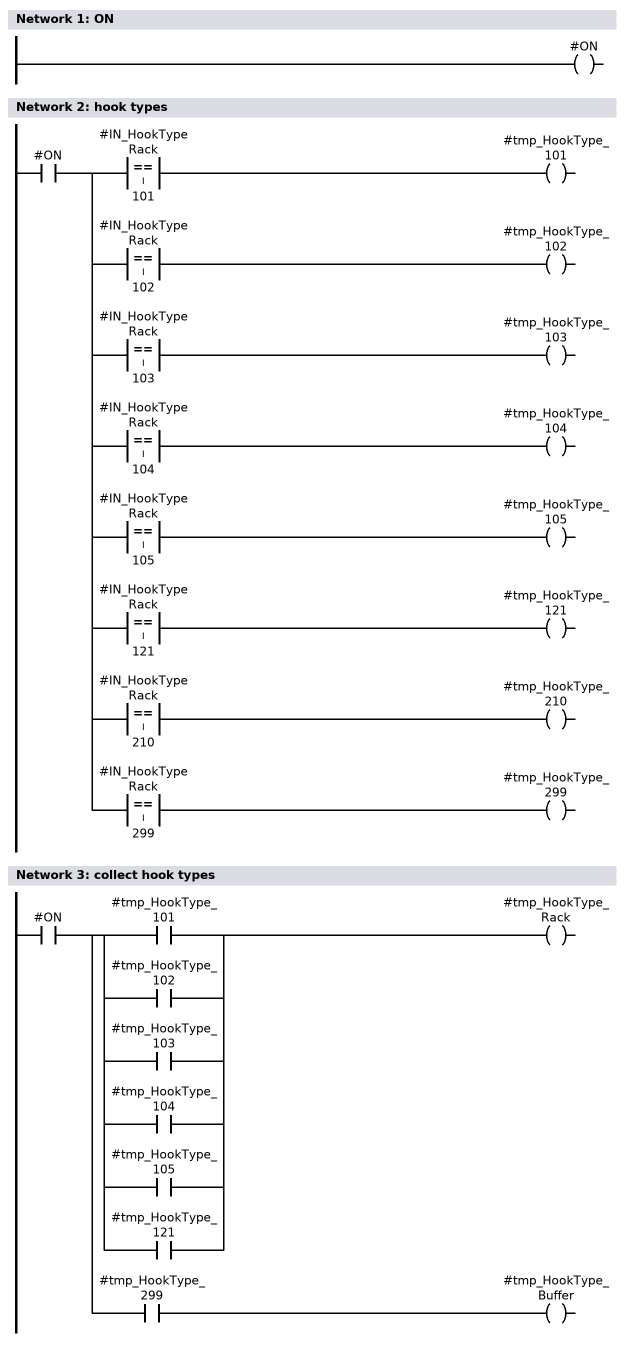
[picture p237: CheckHookType networks 1-3]
NETWORK
TITLE = ON
      SET;
      =     #ON;
NETWORK
TITLE = hook types
      A     #ON;
      =     L 7.0;
      A     L 7.0;
      A(;
      L     #IN_HookTypeRack;
      L     101;
      ==I;
      );
      =     #tmp_HookType_101;
      A     L 7.0;
      A(;
      L     #IN_HookTypeRack;
      L     102;
      ==I;
      );
      =     #tmp_HookType_102;
      A     L 7.0;
      A(;
      L     #IN_HookTypeRack;
      L     103;
      ==I;
      );
      =     #tmp_HookType_103;
      A     L 7.0;
      A(;
      L     #IN_HookTypeRack;
      L     104;
      ==I;
      );
      =     #tmp_HookType_104;
      A     L 7.0;
      A(;
      L     #IN_HookTypeRack;
      L     105;
      ==I;
      );
      =     #tmp_HookType_105;
      A     L 7.0;
      A(;
      L     #IN_HookTypeRack;
      L     121;
      ==I;
      );
      =     #tmp_HookType_121;
      A     L 7.0;
      A(;
      L     #IN_HookTypeRack;
      L     210;
      ==I;
      );
      =     #tmp_HookType_210;
      A     L 7.0;
      A(;
      L     #IN_HookTypeRack;
      L     299;
      ==I;
      );
      =     #tmp_HookType_299;
NETWORK
TITLE = collect hook types
      A     #ON;
      =     L 7.0;
      A     L 7.0;
      A(;
      O     #tmp_HookType_101;
      O     #tmp_HookType_102;
      O     #tmp_HookType_103;
      O     #tmp_HookType_104;
      O     #tmp_HookType_105;
      O     #tmp_HookType_121;
      );
      =     #tmp_HookType_Rack;
      A     L 7.0;
      A     #tmp_HookType_299;
      =     #tmp_HookType_Buffer;
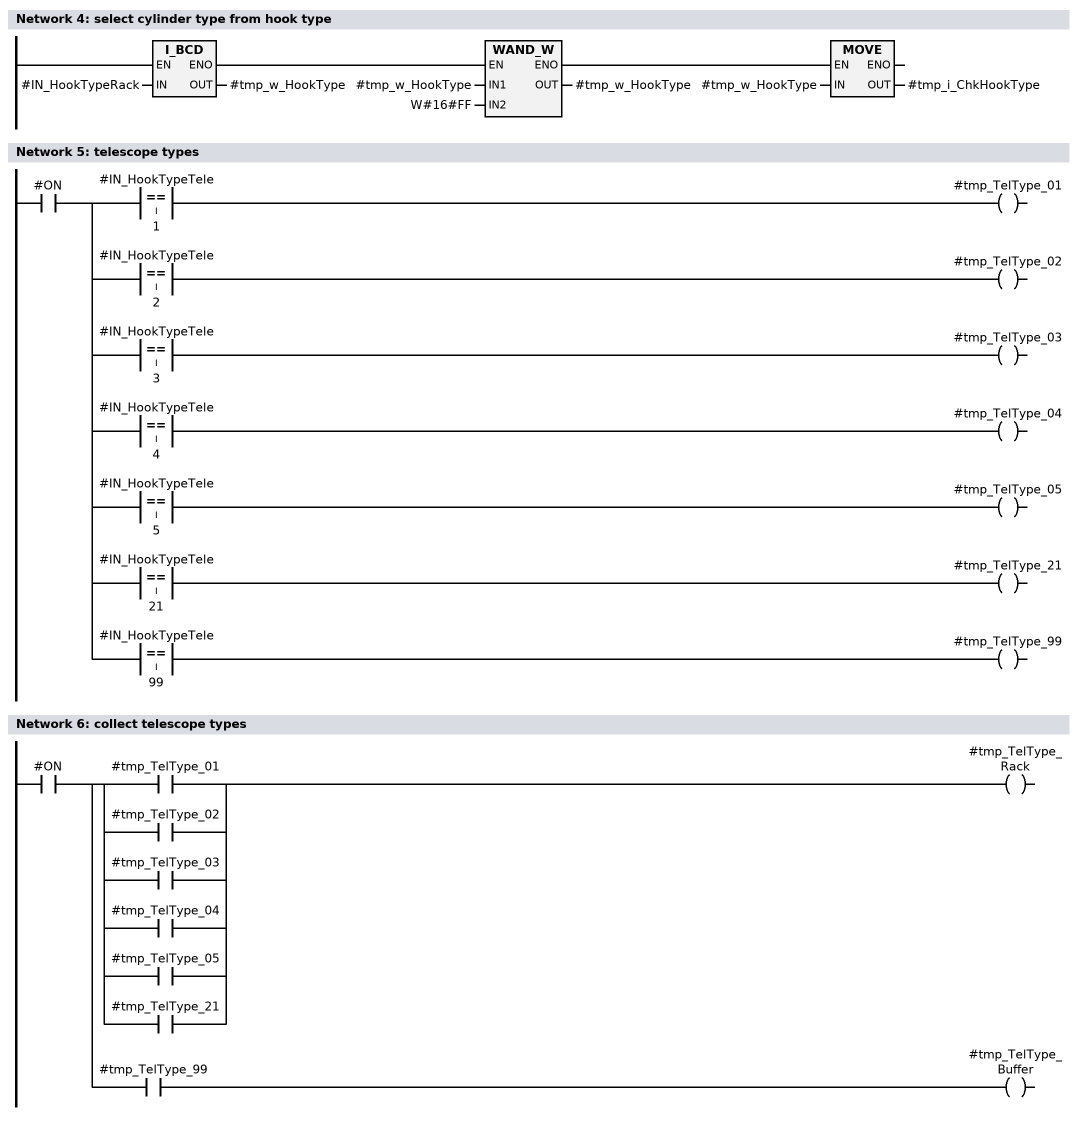
NETWORK
TITLE = select cylinder type from hook type
      A(;
      A(;
      L     #IN_HookTypeRack;
      ITB;
      T     #tmp_w_HookType;
      AN    OV;
      SAVE;
      CLR;
      A     BR;
      );
      JNB   _001;
      L     #tmp_w_HookType;
      L     W#16#FF;
      AW;
      T     #tmp_w_HookType;
      SET;
      SAVE;
      CLR;
_001: A     BR;
      );
      JNB   _002;
      L     #tmp_w_HookType;
      T     #tmp_i_ChkHookType;
_002: NOP   0;
NETWORK
TITLE = telescope types
      A     #ON;
      =     L 7.0;
      A     L 7.0;
      A(;
      L     #IN_HookTypeTele;
      L     1;
      ==I;
      );
      =     #tmp_TelType_01;
      A     L 7.0;
      A(;
      L     #IN_HookTypeTele;
      L     2;
      ==I;
      );
      =     #tmp_TelType_02;
      A     L 7.0;
      A(;
      L     #IN_HookTypeTele;
      L     3;
      ==I;
      );
      =     #tmp_TelType_03;
      A     L 7.0;
      A(;
      L     #IN_HookTypeTele;
      L     4;
      ==I;
      );
      =     #tmp_TelType_04;
      A     L 7.0;
      A(;
      L     #IN_HookTypeTele;
      L     5;
      ==I;
      );
      =     #tmp_TelType_05;
      A     L 7.0;
      A(;
      L     #IN_HookTypeTele;
      L     21;
      ==I;
      );
      =     #tmp_TelType_21;
      A     L 7.0;
      A(;
      L     #IN_HookTypeTele;
      L     99;
      ==I;
      );
      =     #tmp_TelType_99;
NETWORK
TITLE = collect telescope types
      A     #ON;
      =     L 7.0;
      A     L 7.0;
      A(;
      O     #tmp_TelType_01;
      O     #tmp_TelType_02;
      O     #tmp_TelType_03;
      O     #tmp_TelType_04;
      O     #tmp_TelType_05;
      O     #tmp_TelType_21;
      );
      =     #tmp_TelType_Rack;
      A     L 7.0;
      A     #tmp_TelType_99;
      =     #tmp_TelType_Buffer;
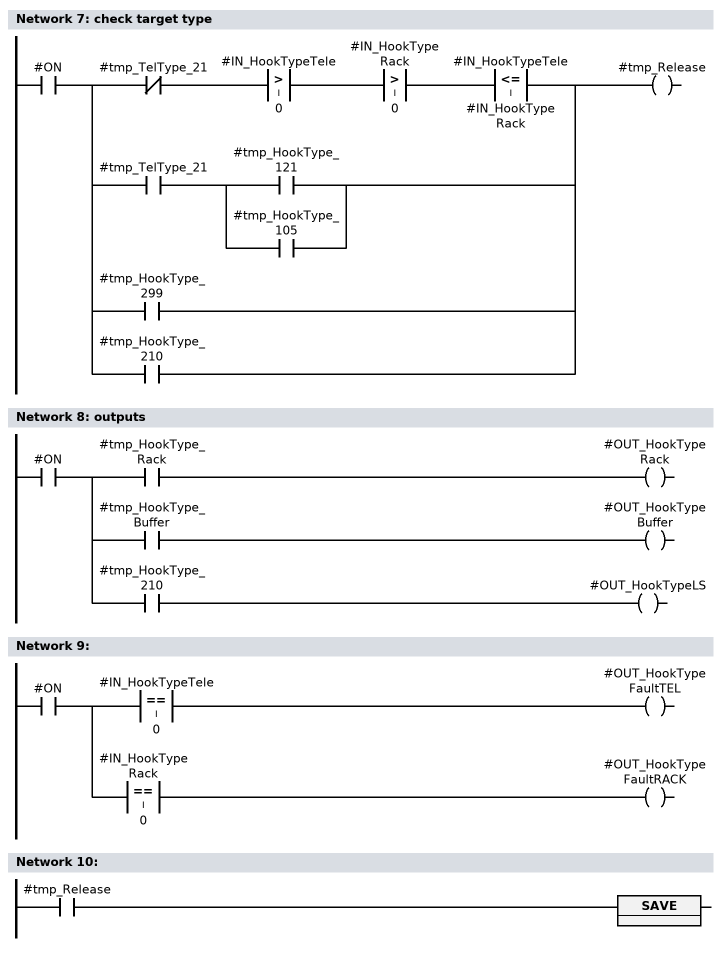
NETWORK
TITLE = check target type
      A     #ON;
      A(;
      AN    #tmp_TelType_21;
      A(;
      L     #IN_HookTypeTele;
      L     0;
      >I;
      );
      A(;
      L     #IN_HookTypeRack;
      L     0;
      >I;
      );
      A(;
      L     #IN_HookTypeTele;
      L     #IN_HookTypeRack;
      <=I;
      );
      O;
      A     #tmp_TelType_21;
      A(;
      O     #tmp_HookType_121;
      O     #tmp_HookType_105;
      );
      O     #tmp_HookType_299;
      O     #tmp_HookType_210;
      );
      =     #tmp_Release;
NETWORK
TITLE = outputs
      A     #ON;
      =     L 7.0;
      A     L 7.0;
      A     #tmp_HookType_Rack;
      =     #OUT_HookTypeRack;
      A     L 7.0;
      A     #tmp_HookType_Buffer;
      =     #OUT_HookTypeBuffer;
      A     L 7.0;
      A     #tmp_HookType_210;
      =     #OUT_HookTypeLS;
NETWORK
TITLE =
      A     #ON;
      =     L 7.0;
      A     L 7.0;
      A(;
      L     #IN_HookTypeTele;
      L     0;
      ==I;
      );
      =     #OUT_HookTypeFaultTEL;
      A     L 7.0;
      A(;
      L     #IN_HookTypeRack;
      L     0;
      ==I;
      );
      =     #OUT_HookTypeFaultRACK;
NETWORK
TITLE =
      A     #tmp_Release;
      SAVE;
END_FUNCTION

FUNCTION "CheckWindowDi" : VOID	// FC 100
TITLE = Check Window
VERSION : 1.0
VAR_INPUT
  IN_diValue : DINT ;
  IN_diTestFor : DINT ;
  IN_diTolMinus : DINT ;
  IN_diTolPlus : DINT ;
END_VAR
VAR_OUTPUT
  OUT_xInWindow : BOOL ;
  OUT_udiAbsDiff : DINT ;
END_VAR
VAR_TEMP
  INT_diWinMinus : DINT ;
  INT_diWinPlus : DINT ;
  INT_xInWindow : BOOL ;
END_VAR
BEGIN
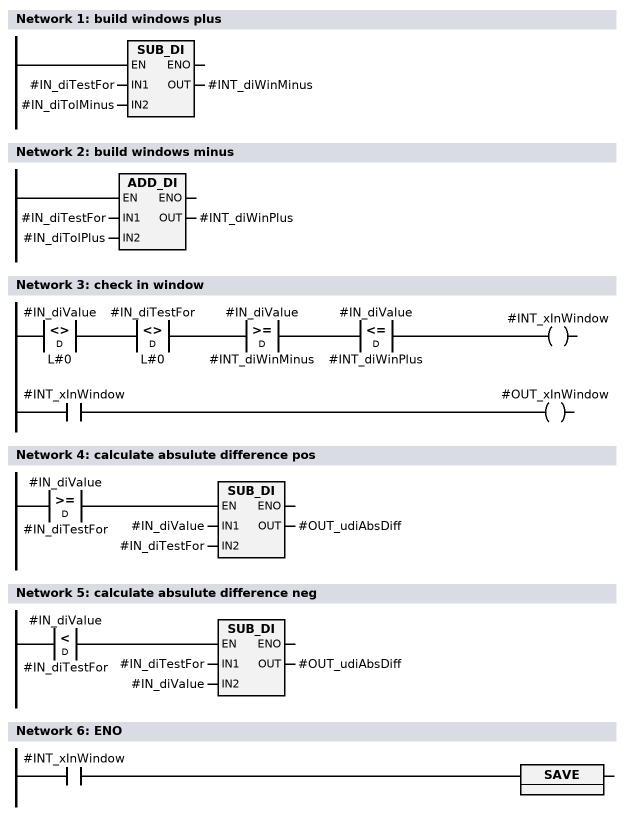
NETWORK
TITLE = build windows plus
      L     #IN_diTestFor;
      L     #IN_diTolMinus;
      -D;
      T     #INT_diWinMinus;
      NOP   0;
NETWORK
TITLE = build windows minus
      L     #IN_diTestFor;
      L     #IN_diTolPlus;
      +D;
      T     #INT_diWinPlus;
      NOP   0;
NETWORK
TITLE = check in window
      A(;
      L     #IN_diValue;
      L     L#0;
      <>D;
      );
      A(;
      L     #IN_diTestFor;
      L     L#0;
      <>D;
      );
      A(;
      L     #IN_diValue;
      L     #INT_diWinMinus;
      >=D;
      );
      A(;
      L     #IN_diValue;
      L     #INT_diWinPlus;
      <=D;
      );
      =     #INT_xInWindow;
      A     #INT_xInWindow;
      =     #OUT_xInWindow;
NETWORK
TITLE = calculate absulute difference pos
      A(;
      L     #IN_diValue;
      L     #IN_diTestFor;
      >=D;
      );
      JNB   _001;
      L     #IN_diValue;
      L     #IN_diTestFor;
      -D;
      T     #OUT_udiAbsDiff;
_001: NOP   0;
NETWORK
TITLE = calculate absulute difference neg
      A(;
      L     #IN_diValue;
      L     #IN_diTestFor;
      <D;
      );
      JNB   _002;
      L     #IN_diTestFor;
      L     #IN_diValue;
      -D;
      T     #OUT_udiAbsDiff;
_002: NOP   0;
NETWORK
TITLE = ENO
      A     #INT_xInWindow;
      SAVE;
END_FUNCTION

FUNCTION "Communication" : VOID	// FC 103
VERSION : 0.1
VAR_TEMP
  tmp_result : INT ;
  rel_online : BOOL ;
  val : DINT ;
END_VAR
BEGIN
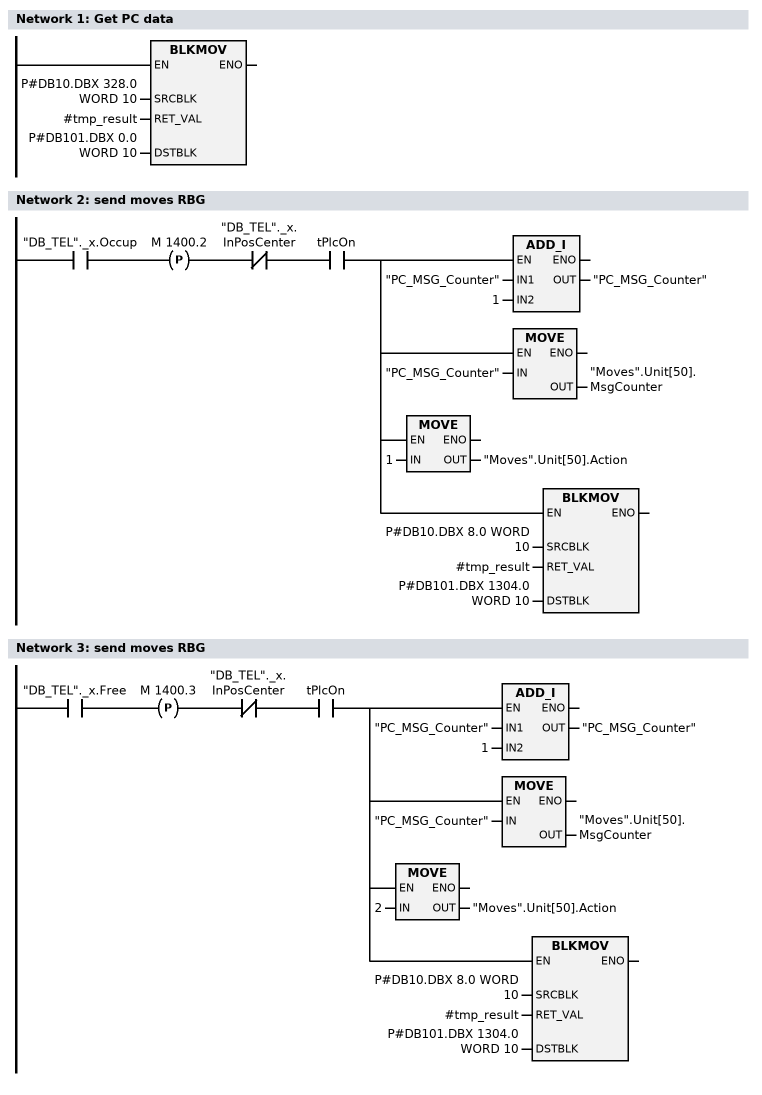
NETWORK
TITLE = Get PC data
      CALL  "BLKMOV" (
           SRCBLK                   := P#DB10.DBX 328.0 WORD 10,
           RET_VAL                  := #tmp_result,
           DSTBLK                   := P#DB101.DBX 0.0 WORD 10);
      NOP   0;
NETWORK
TITLE = send moves RBG
//Telescopes occupied
      A     "DB_TEL"._x.Occup;
      FP    M 1400.2;
      AN    "DB_TEL"._x.InPosCenter;
      A     "tPlcOn";
      =     L 8.0;
      A     L 8.0;
      JNB   _001;
      L     "PC_MSG_Counter";
      L     1;
      +I;
      T     "PC_MSG_Counter";
_001: NOP   0;
      A     L 8.0;
      JNB   _002;
      L     "PC_MSG_Counter";
      T     "Moves".Unit[50].MsgCounter;
_002: NOP   0;
      A     L 8.0;
      JNB   _003;
      L     1;
      T     "Moves".Unit[50].Action;
_003: NOP   0;
      A     L 8.0;
      JNB   _004;
      CALL  "BLKMOV" (
           SRCBLK                   := P#DB10.DBX 8.0 WORD 10,
           RET_VAL                  := #tmp_result,
           DSTBLK                   := P#DB101.DBX 1304.0 WORD 10);
_004: NOP   0;
NETWORK
TITLE = send moves RBG
//Telescopes empty
      A     "DB_TEL"._x.Free;
      FP    M 1400.3;
      AN    "DB_TEL"._x.InPosCenter;
      A     "tPlcOn";
      =     L 8.0;
      A     L 8.0;
      JNB   _005;
      L     "PC_MSG_Counter";
      L     1;
      +I;
      T     "PC_MSG_Counter";
_005: NOP   0;
      A     L 8.0;
      JNB   _006;
      L     "PC_MSG_Counter";
      T     "Moves".Unit[50].MsgCounter;
_006: NOP   0;
      A     L 8.0;
      JNB   _007;
      L     2;
      T     "Moves".Unit[50].Action;
_007: NOP   0;
      A     L 8.0;
      JNB   _008;
      CALL  "BLKMOV" (
           SRCBLK                   := P#DB10.DBX 8.0 WORD 10,
           RET_VAL                  := #tmp_result,
           DSTBLK                   := P#DB101.DBX 1304.0 WORD 10);
_008: NOP   0;
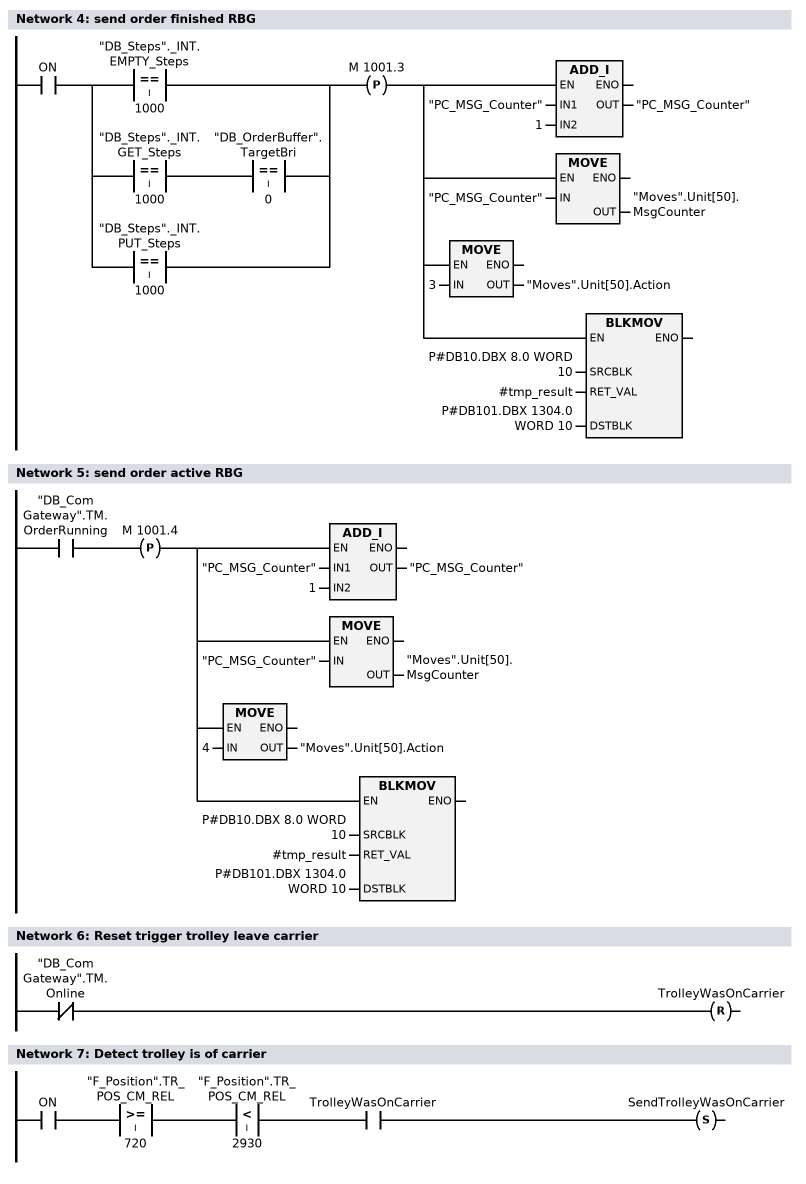
NETWORK
TITLE = send order finished RBG
      A     "ON";
      A(;
      O(;
      L     "DB_Steps"._INT.EMPTY_Steps;
      L     1000;
      ==I;
      );
      O;
      A(;
      L     "DB_Steps"._INT.GET_Steps;
      L     1000;
      ==I;
      );
      A(;
      L     "DB_OrderBuffer".TargetBri;
      L     0;
      ==I;
      );
      O(;
      L     "DB_Steps"._INT.PUT_Steps;
      L     1000;
      ==I;
      );
      );
      FP    M 1001.3;
      =     L 8.0;
      A     L 8.0;
      JNB   _009;
      L     "PC_MSG_Counter";
      L     1;
      +I;
      T     "PC_MSG_Counter";
_009: NOP   0;
      A     L 8.0;
      JNB   _00a;
      L     "PC_MSG_Counter";
      T     "Moves".Unit[50].MsgCounter;
_00a: NOP   0;
      A     L 8.0;
      JNB   _00b;
      L     3;
      T     "Moves".Unit[50].Action;
_00b: NOP   0;
      A     L 8.0;
      JNB   _00c;
      CALL  "BLKMOV" (
           SRCBLK                   := P#DB10.DBX 8.0 WORD 10,
           RET_VAL                  := #tmp_result,
           DSTBLK                   := P#DB101.DBX 1304.0 WORD 10);
_00c: NOP   0;
NETWORK
TITLE = send order active RBG
      A     "DB_ComGateway".TM.OrderRunning;
      FP    M 1001.4;
      =     L 8.0;
      A     L 8.0;
      JNB   _00d;
      L     "PC_MSG_Counter";
      L     1;
      +I;
      T     "PC_MSG_Counter";
_00d: NOP   0;
      A     L 8.0;
      JNB   _00e;
      L     "PC_MSG_Counter";
      T     "Moves".Unit[50].MsgCounter;
_00e: NOP   0;
      A     L 8.0;
      JNB   _00f;
      L     4;
      T     "Moves".Unit[50].Action;
_00f: NOP   0;
      A     L 8.0;
      JNB   _010;
      CALL  "BLKMOV" (
           SRCBLK                   := P#DB10.DBX 8.0 WORD 10,
           RET_VAL                  := #tmp_result,
           DSTBLK                   := P#DB101.DBX 1304.0 WORD 10);
_010: NOP   0;
NETWORK
TITLE = Reset trigger trolley leave carrier
      AN    "DB_ComGateway".TM.Online;
      R     "TrolleyWasOnCarrier";
NETWORK
TITLE = Detect trolley is of carrier
      A     "ON";
      A(;
      L     "F_Position".TR_POS_CM_REL;
      L     720;
      >=I;
      );
      A(;
      L     "F_Position".TR_POS_CM_REL;
      L     2930;
      <I;
      );
      A     "TrolleyWasOnCarrier";
      S     "SendTrolleyWasOnCarrier";
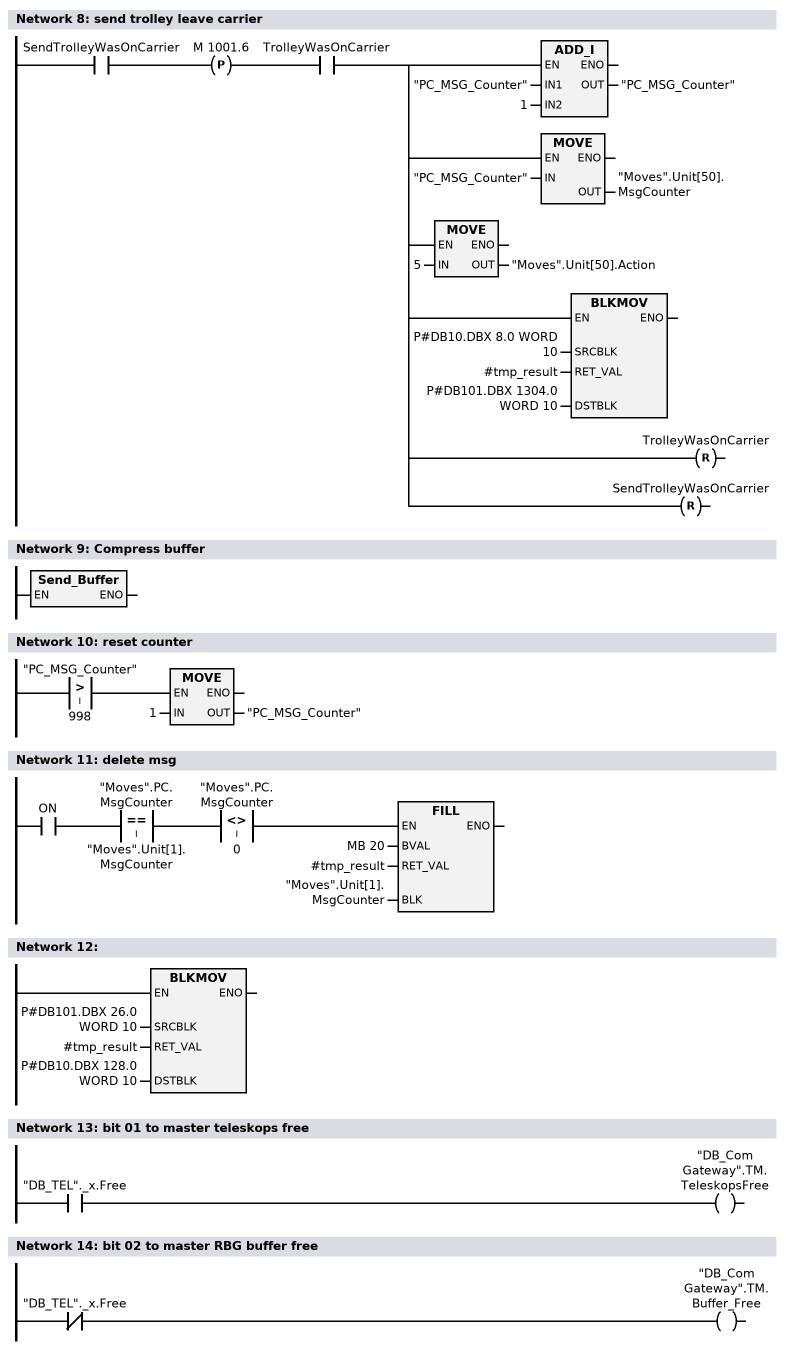
NETWORK
TITLE = send trolley leave carrier
      A     "SendTrolleyWasOnCarrier";
      FP    M 1001.6;
      A     "TrolleyWasOnCarrier";
      =     L 8.0;
      A     L 8.0;
      JNB   _011;
      L     "PC_MSG_Counter";
      L     1;
      +I;
      T     "PC_MSG_Counter";
_011: NOP   0;
      A     L 8.0;
      JNB   _012;
      L     "PC_MSG_Counter";
      T     "Moves".Unit[50].MsgCounter;
_012: NOP   0;
      A     L 8.0;
      JNB   _013;
      L     5;
      T     "Moves".Unit[50].Action;
_013: NOP   0;
      A     L 8.0;
      JNB   _014;
      CALL  "BLKMOV" (
           SRCBLK                   := P#DB10.DBX 8.0 WORD 10,
           RET_VAL                  := #tmp_result,
           DSTBLK                   := P#DB101.DBX 1304.0 WORD 10);
_014: NOP   0;
      A     L 8.0;
      BLD   102;
      R     "TrolleyWasOnCarrier";
      A     L 8.0;
      BLD   102;
      R     "SendTrolleyWasOnCarrier";
NETWORK
TITLE = Compress buffer
      CALL  "Send_Buffer";
      NOP   0;
NETWORK
TITLE = reset counter
      A(;
      L     "PC_MSG_Counter";
      L     998;
      >I;
      );
      JNB   _015;
      L     1;
      T     "PC_MSG_Counter";
_015: NOP   0;
NETWORK
TITLE = delete msg
      A     "ON";
      A(;
      L     "Moves".PC.MsgCounter;
      L     "Moves".Unit[1].MsgCounter;
      ==I;
      );
      A(;
      L     "Moves".PC.MsgCounter;
      L     0;
      <>I;
      );
      JNB   _016;
      CALL  "FILL" (
           BVAL                     := MB 20,
           RET_VAL                  := #tmp_result,
           BLK                      := "Moves".Unit[1].MsgCounter);
_016: NOP   0;
NETWORK
TITLE =
      CALL  "BLKMOV" (
           SRCBLK                   := P#DB101.DBX 26.0 WORD 10,
           RET_VAL                  := #tmp_result,
           DSTBLK                   := P#DB10.DBX 128.0 WORD 10);
      NOP   0;
NETWORK
TITLE = bit 01 to master teleskops free
      A     "DB_TEL"._x.Free;
      =     "DB_ComGateway".TM.TeleskopsFree;
NETWORK
TITLE = bit 02 to master RBG buffer free
      AN    "DB_TEL"._x.Free;
      =     "DB_ComGateway".TM.Buffer_Free;
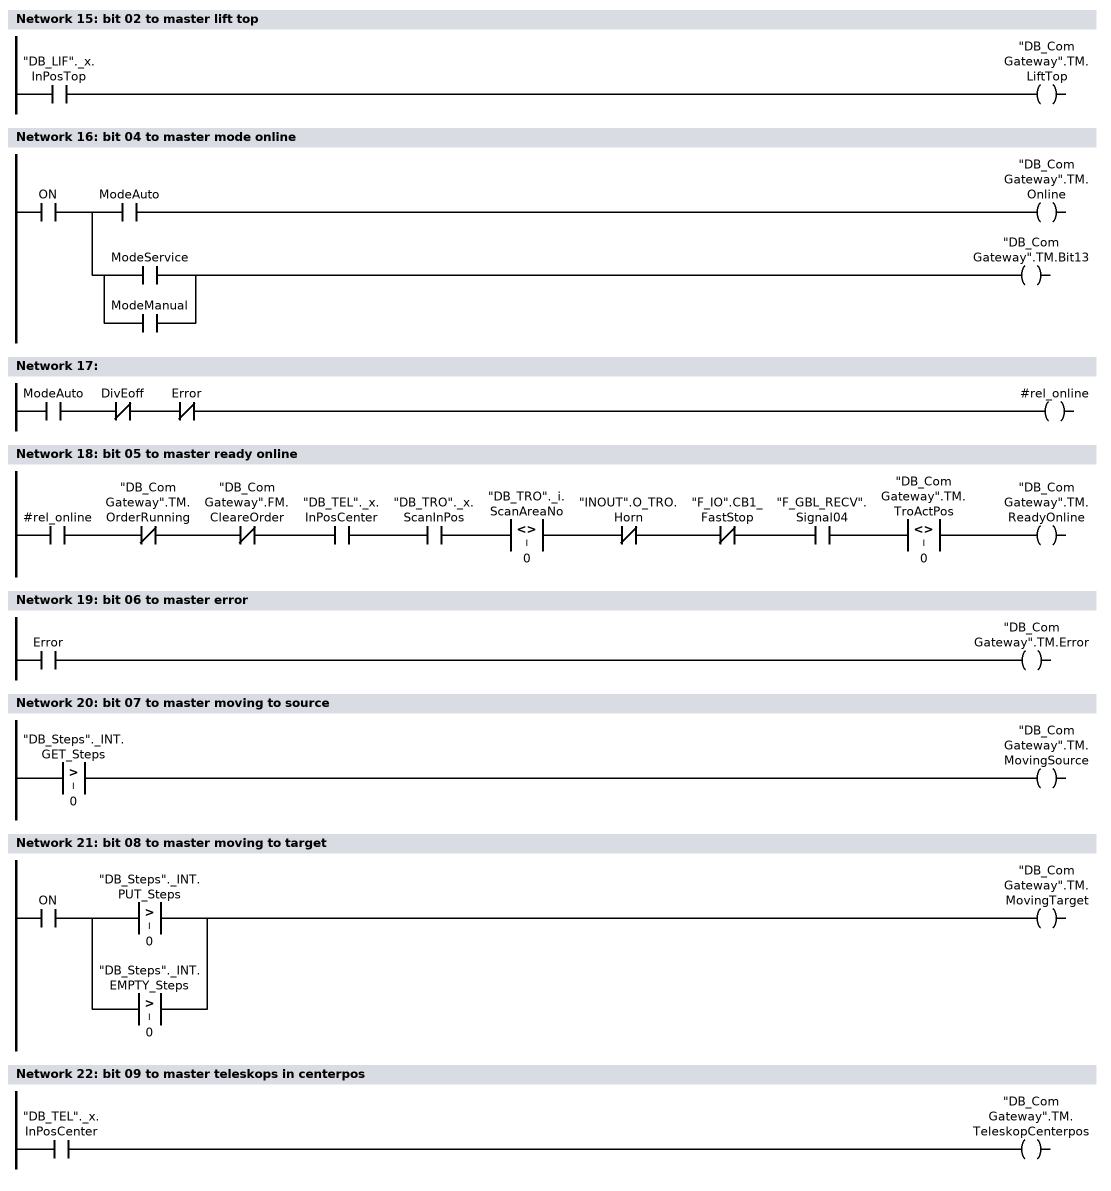
NETWORK
TITLE = bit 02 to master lift top
      A     "DB_LIF"._x.InPosTop;
      =     "DB_ComGateway".TM.LiftTop;
NETWORK
TITLE = bit 04 to master mode online
      A     "ON";
      =     L 8.0;
      A     L 8.0;
      A     "ModeAuto";
      =     "DB_ComGateway".TM.Online;
      A     L 8.0;
      A(;
      O     "ModeService";
      O     "ModeManual";
      );
      =     "DB_ComGateway".TM.Bit13;
NETWORK
TITLE =
      A     "ModeAuto";
      AN    "DivEoff";
      AN    "Error";
      =     #rel_online;
NETWORK
TITLE = bit 05 to master ready online
      A     #rel_online;
      AN    "DB_ComGateway".TM.OrderRunning;
      AN    "DB_ComGateway".FM.CleareOrder;
      A     "DB_TEL"._x.InPosCenter;
      A     "DB_TRO"._x.ScanInPos;
      A(;
      L     "DB_TRO"._i.ScanAreaNo;
      L     0;
      <>I;
      );
      AN    "INOUT".O_TRO.Horn;
      AN    "F_IO".CB1_FastStop;
      A     "F_GBL_RECV".Signal04;
      A(;
      L     "DB_ComGateway".TM.TroActPos;
      L     0;
      <>I;
      );
      =     "DB_ComGateway".TM.ReadyOnline;
NETWORK
TITLE = bit 06 to master error
      A     "Error";
      =     "DB_ComGateway".TM.Error;
NETWORK
TITLE = bit 07 to master moving to source
      L     "DB_Steps"._INT.GET_Steps;
      L     0;
      >I;
      =     "DB_ComGateway".TM.MovingSource;
NETWORK
TITLE = bit 08 to master moving to target
      A     "ON";
      A(;
      O(;
      L     "DB_Steps"._INT.PUT_Steps;
      L     0;
      >I;
      );
      O(;
      L     "DB_Steps"._INT.EMPTY_Steps;
      L     0;
      >I;
      );
      );
      =     "DB_ComGateway".TM.MovingTarget;
NETWORK
TITLE = bit 09 to master teleskops in centerpos
      A     "DB_TEL"._x.InPosCenter;
      =     "DB_ComGateway".TM.TeleskopCenterpos;
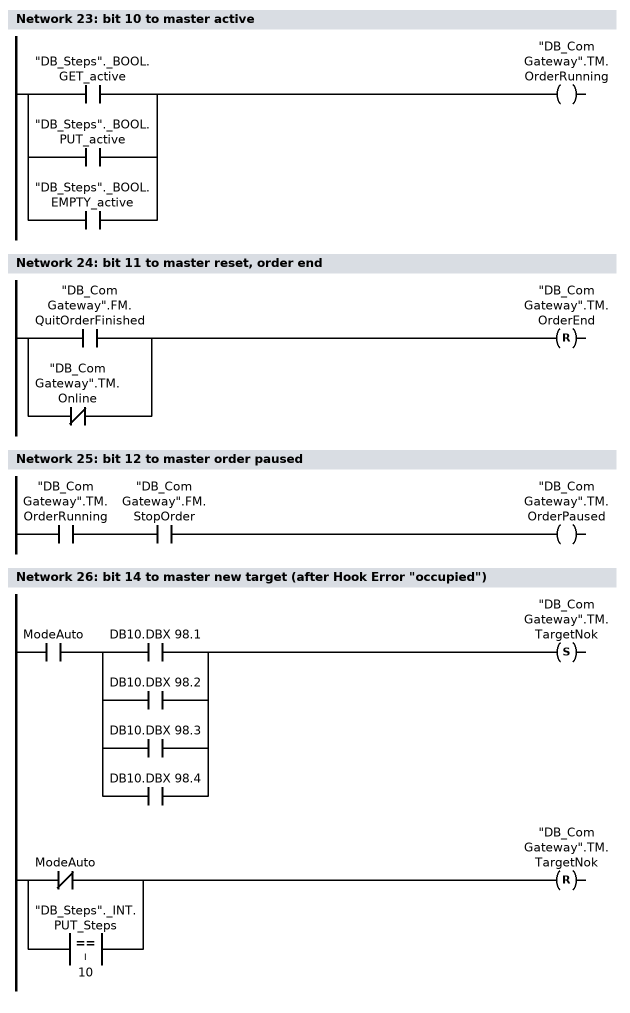
NETWORK
TITLE = bit 10 to master active
      O     "DB_Steps"._BOOL.GET_active;
      O     "DB_Steps"._BOOL.PUT_active;
      O     "DB_Steps"._BOOL.EMPTY_active;
      =     "DB_ComGateway".TM.OrderRunning;
NETWORK
TITLE = bit 11 to master reset, order end
      O     "DB_ComGateway".FM.QuitOrderFinished;
      ON    "DB_ComGateway".TM.Online;
      R     "DB_ComGateway".TM.OrderEnd;
NETWORK
TITLE = bit 12 to master order paused
      A     "DB_ComGateway".TM.OrderRunning;
      A     "DB_ComGateway".FM.StopOrder;
      =     "DB_ComGateway".TM.OrderPaused;
NETWORK
TITLE = bit 14 to master new target (after Hook Error "occupied")
//New Target:
//
      A     "ModeAuto";
      A(;
      O     DB10.DBX 98.1;
      O     DB10.DBX 98.2;
      O     DB10.DBX 98.3;
      O     DB10.DBX 98.4;
      );
      S     "DB_ComGateway".TM.TargetNok;
      A(;
      ON    "ModeAuto";
      O(;
      L     "DB_Steps"._INT.PUT_Steps;
      L     10;
      ==I;
      );
      );
      R     "DB_ComGateway".TM.TargetNok;
      NOP   0;
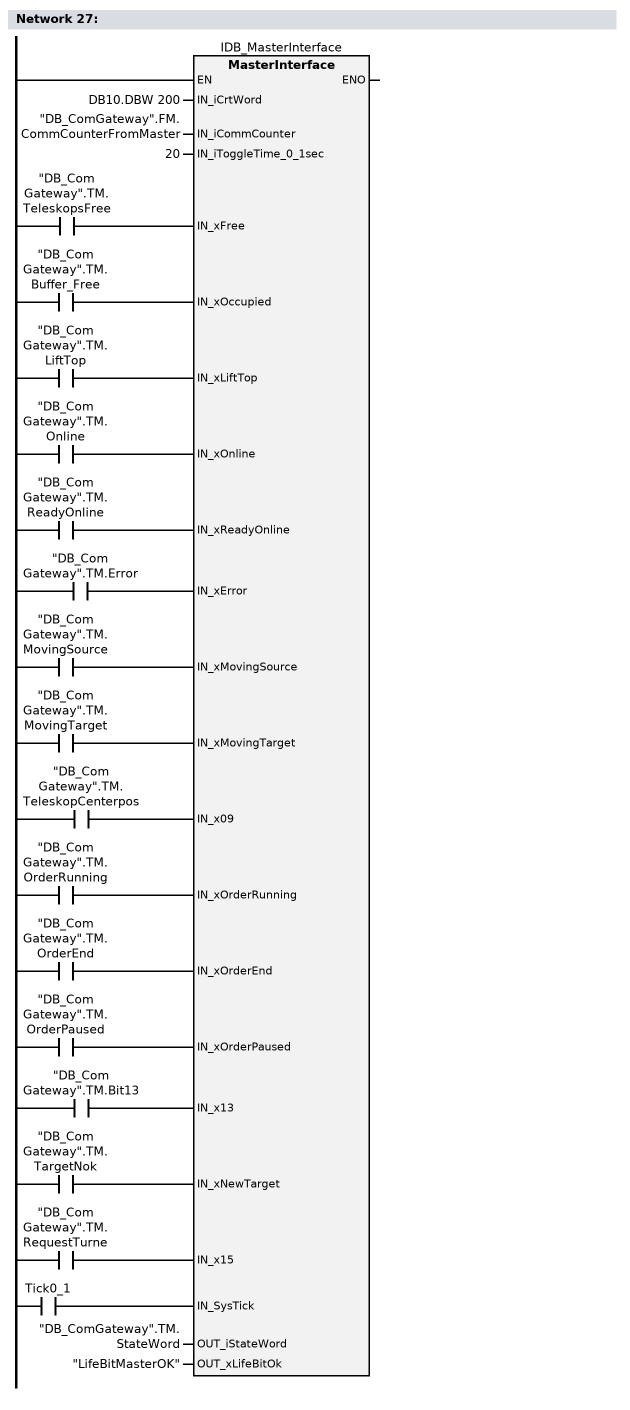
NETWORK
TITLE =
//we do not need the outputs....
//
      A     "DB_ComGateway".TM.TeleskopsFree;
      =     L 8.0;
      BLD   103;
      A     "DB_ComGateway".TM.Buffer_Free;
      =     L 8.1;
      BLD   103;
      A     "DB_ComGateway".TM.LiftTop;
      =     L 8.2;
      BLD   103;
      A     "DB_ComGateway".TM.Online;
      =     L 8.3;
      BLD   103;
      A     "DB_ComGateway".TM.ReadyOnline;
      =     L 8.4;
      BLD   103;
      A     "DB_ComGateway".TM.Error;
      =     L 8.5;
      BLD   103;
      A     "DB_ComGateway".TM.MovingSource;
      =     L 8.6;
      BLD   103;
      A     "DB_ComGateway".TM.MovingTarget;
      =     L 8.7;
      BLD   103;
      A     "DB_ComGateway".TM.TeleskopCenterpos;
      =     L 9.0;
      BLD   103;
      A     "DB_ComGateway".TM.OrderRunning;
      =     L 9.1;
      BLD   103;
      A     "DB_ComGateway".TM.OrderEnd;
      =     L 9.2;
      BLD   103;
      A     "DB_ComGateway".TM.OrderPaused;
      =     L 9.3;
      BLD   103;
      A     "DB_ComGateway".TM.Bit13;
      =     L 9.4;
      BLD   103;
      A     "DB_ComGateway".TM.TargetNok;
      =     L 9.5;
      BLD   103;
      A     "DB_ComGateway".TM.RequestTurne;
      =     L 9.6;
      BLD   103;
      A     "Tick0_1";
      =     L 9.7;
      BLD   103;
      CALL  "MasterInterface" , "IDB_MasterInterface" (
           IN_iCrtWord              := DB10.DBW 200,
           IN_iCommCounter          := "DB_ComGateway".FM.CommCounterFromMaster,
           IN_iToggleTime_0_1sec    := 20,
           IN_xFree                 := L 8.0,
           IN_xOccupied             := L 8.1,
           IN_xLiftTop              := L 8.2,
           IN_xOnline               := L 8.3,
           IN_xReadyOnline          := L 8.4,
           IN_xError                := L 8.5,
           IN_xMovingSource         := L 8.6,
           IN_xMovingTarget         := L 8.7,
           IN_x09                   := L 9.0,
           IN_xOrderRunning         := L 9.1,
           IN_xOrderEnd             := L 9.2,
           IN_xOrderPaused          := L 9.3,
           IN_x13                   := L 9.4,
           IN_xNewTarget            := L 9.5,
           IN_x15                   := L 9.6,
           IN_SysTick               := L 9.7,
           OUT_iStateWord           := "DB_ComGateway".TM.StateWord,
           OUT_xLifeBitOk           := "LifeBitMasterOK");
      NOP   0;
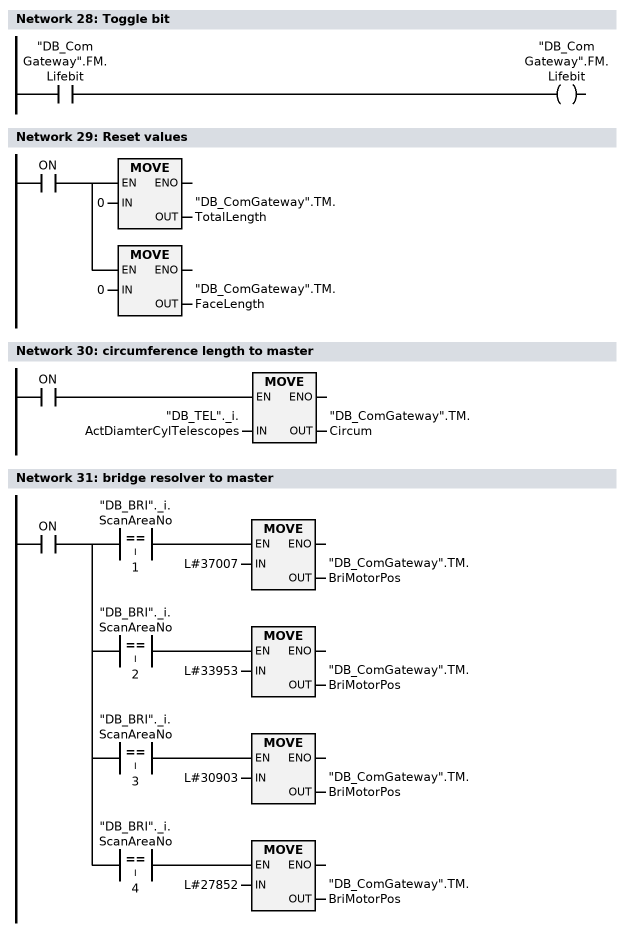
NETWORK
TITLE = Toggle bit
      A     "DB_ComGateway".FM.Lifebit;
      =     "DB_ComGateway".FM.Lifebit;
NETWORK
TITLE = Reset values
      A     "ON";
      =     L 8.0;
      A     L 8.0;
      JNB   _017;
      L     0;
      T     "DB_ComGateway".TM.TotalLength;
_017: NOP   0;
      A     L 8.0;
      JNB   _018;
      L     0;
      T     "DB_ComGateway".TM.FaceLength;
_018: NOP   0;
NETWORK
TITLE = circumference length to master
      A     "ON";
      JNB   _019;
      L     "DB_TEL"._i.ActDiamterCylTelescopes;
      T     "DB_ComGateway".TM.Circum;
_019: NOP   0;
NETWORK
TITLE = bridge resolver to master
      A     "ON";
      =     L 8.0;
      A     L 8.0;
      A(;
      L     "DB_BRI"._i.ScanAreaNo;
      L     1;
      ==I;
      );
      JNB   _01a;
      L     L#37007;
      T     "DB_ComGateway".TM.BriMotorPos;
_01a: NOP   0;
      A     L 8.0;
      A(;
      L     "DB_BRI"._i.ScanAreaNo;
      L     2;
      ==I;
      );
      JNB   _01b;
      L     L#33953;
      T     "DB_ComGateway".TM.BriMotorPos;
_01b: NOP   0;
      A     L 8.0;
      A(;
      L     "DB_BRI"._i.ScanAreaNo;
      L     3;
      ==I;
      );
      JNB   _01c;
      L     L#30903;
      T     "DB_ComGateway".TM.BriMotorPos;
_01c: NOP   0;
      A     L 8.0;
      A(;
      L     "DB_BRI"._i.ScanAreaNo;
      L     4;
      ==I;
      );
      JNB   _01d;
      L     L#27852;
      T     "DB_ComGateway".TM.BriMotorPos;
_01d: NOP   0;
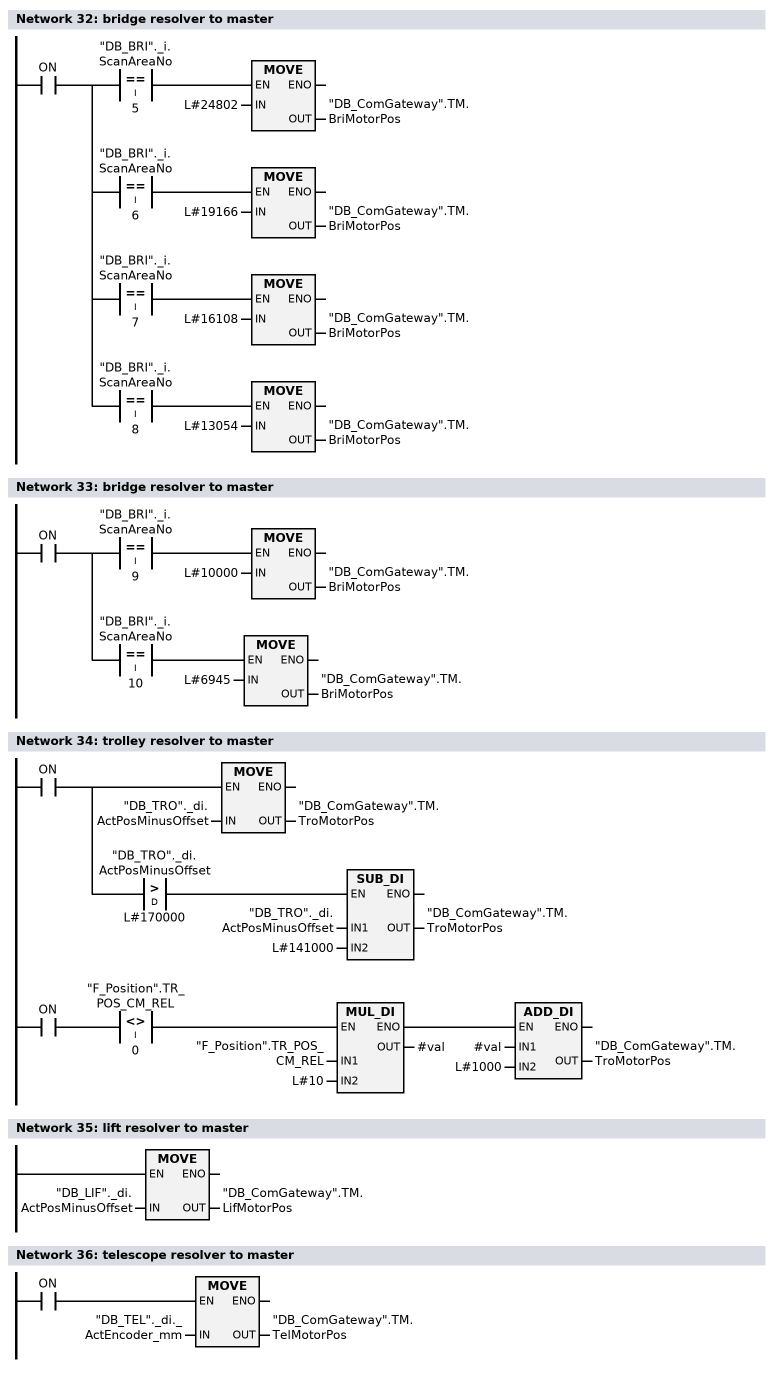
NETWORK
TITLE = bridge resolver to master
      A     "ON";
      =     L 8.0;
      A     L 8.0;
      A(;
      L     "DB_BRI"._i.ScanAreaNo;
      L     5;
      ==I;
      );
      JNB   _01e;
      L     L#24802;
      T     "DB_ComGateway".TM.BriMotorPos;
_01e: NOP   0;
      A     L 8.0;
      A(;
      L     "DB_BRI"._i.ScanAreaNo;
      L     6;
      ==I;
      );
      JNB   _01f;
      L     L#19166;
      T     "DB_ComGateway".TM.BriMotorPos;
_01f: NOP   0;
      A     L 8.0;
      A(;
      L     "DB_BRI"._i.ScanAreaNo;
      L     7;
      ==I;
      );
      JNB   _020;
      L     L#16108;
      T     "DB_ComGateway".TM.BriMotorPos;
_020: NOP   0;
      A     L 8.0;
      A(;
      L     "DB_BRI"._i.ScanAreaNo;
      L     8;
      ==I;
      );
      JNB   _021;
      L     L#13054;
      T     "DB_ComGateway".TM.BriMotorPos;
_021: NOP   0;
NETWORK
TITLE = bridge resolver to master
      A     "ON";
      =     L 8.0;
      A     L 8.0;
      A(;
      L     "DB_BRI"._i.ScanAreaNo;
      L     9;
      ==I;
      );
      JNB   _022;
      L     L#10000;
      T     "DB_ComGateway".TM.BriMotorPos;
_022: NOP   0;
      A     L 8.0;
      A(;
      L     "DB_BRI"._i.ScanAreaNo;
      L     10;
      ==I;
      );
      JNB   _023;
      L     L#6945;
      T     "DB_ComGateway".TM.BriMotorPos;
_023: NOP   0;
NETWORK
TITLE = trolley resolver to master
      A     "ON";
      =     L 8.0;
      A     L 8.0;
      JNB   _024;
      L     "DB_TRO"._di.ActPosMinusOffset;
      T     "DB_ComGateway".TM.TroMotorPos;
_024: NOP   0;
      A(;
      A     L 8.0;
      A(;
      L     "F_Position".TR_POS_CM_REL;
      L     0;
      <>I;
      );
      JNB   _025;
      L     "F_Position".TR_POS_CM_REL;
      L     L#10;
      *D;
      T     #val;
      AN    OV;
      SAVE;
      CLR;
_025: A     BR;
      );
      JNB   _026;
      L     #val;
      L     L#1000;
      +D;
      T     "DB_ComGateway".TM.TroMotorPos;
_026: NOP   0;
      A     L 8.0;
      A(;
      L     "DB_TRO"._di.ActPosMinusOffset;
      L     L#170000;
      >D;
      );
      JNB   _027;
      L     "DB_TRO"._di.ActPosMinusOffset;
      L     L#141000;
      -D;
      T     "DB_ComGateway".TM.TroMotorPos;
_027: NOP   0;
NETWORK
TITLE = lift resolver to master
      L     "DB_LIF"._di.ActPosMinusOffset;
      T     "DB_ComGateway".TM.LifMotorPos;
      NOP   0;
NETWORK
TITLE = telescope resolver to master
      A     "ON";
      JNB   _028;
      L     "DB_TEL"._di._ActEncoder_mm;
      T     "DB_ComGateway".TM.TelMotorPos;
_028: NOP   0;
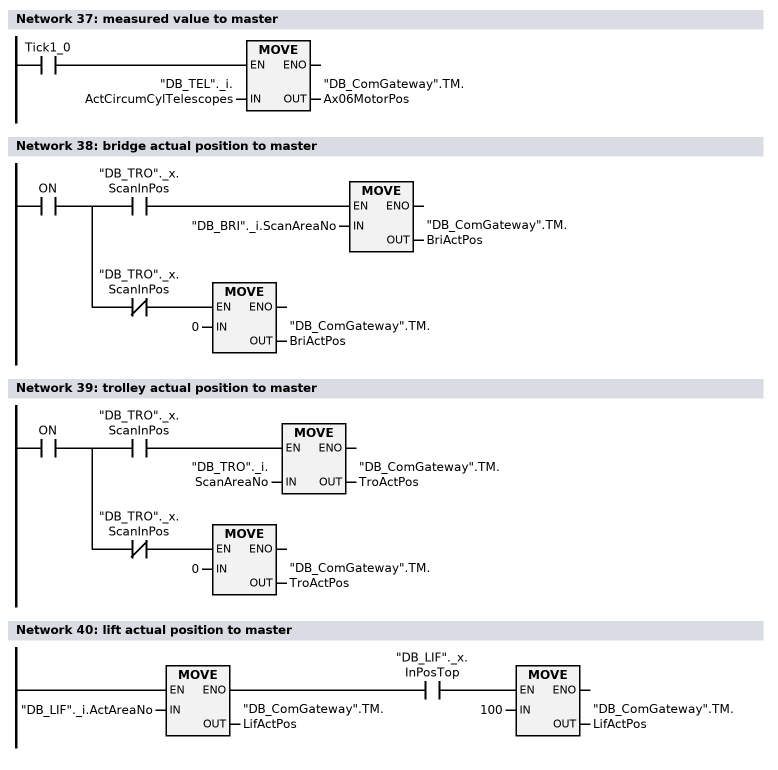
NETWORK
TITLE = measured value to master
      A     "Tick1_0";
      JNB   _029;
      L     "DB_TEL"._i.ActCircumCylTelescopes;
      T     "DB_ComGateway".TM.Ax06MotorPos;
_029: NOP   0;
NETWORK
TITLE = bridge actual position to master
      A     "ON";
      =     L 8.0;
      A     L 8.0;
      A     "DB_TRO"._x.ScanInPos;
      JNB   _02a;
      L     "DB_BRI"._i.ScanAreaNo;
      T     "DB_ComGateway".TM.BriActPos;
_02a: NOP   0;
      A     L 8.0;
      AN    "DB_TRO"._x.ScanInPos;
      JNB   _02b;
      L     0;
      T     "DB_ComGateway".TM.BriActPos;
_02b: NOP   0;
NETWORK
TITLE = trolley actual position to master
      A     "ON";
      =     L 8.0;
      A     L 8.0;
      A     "DB_TRO"._x.ScanInPos;
      JNB   _02c;
      L     "DB_TRO"._i.ScanAreaNo;
      T     "DB_ComGateway".TM.TroActPos;
_02c: NOP   0;
      A     L 8.0;
      AN    "DB_TRO"._x.ScanInPos;
      JNB   _02d;
      L     0;
      T     "DB_ComGateway".TM.TroActPos;
_02d: NOP   0;
NETWORK
TITLE = lift actual position to master
      A(;
      L     "DB_LIF"._i.ActAreaNo;
      T     "DB_ComGateway".TM.LifActPos;
      SET;
      SAVE;
      CLR;
      A     BR;
      );
      A     "DB_LIF"._x.InPosTop;
      JNB   _02e;
      L     100;
      T     "DB_ComGateway".TM.LifActPos;
_02e: NOP   0;
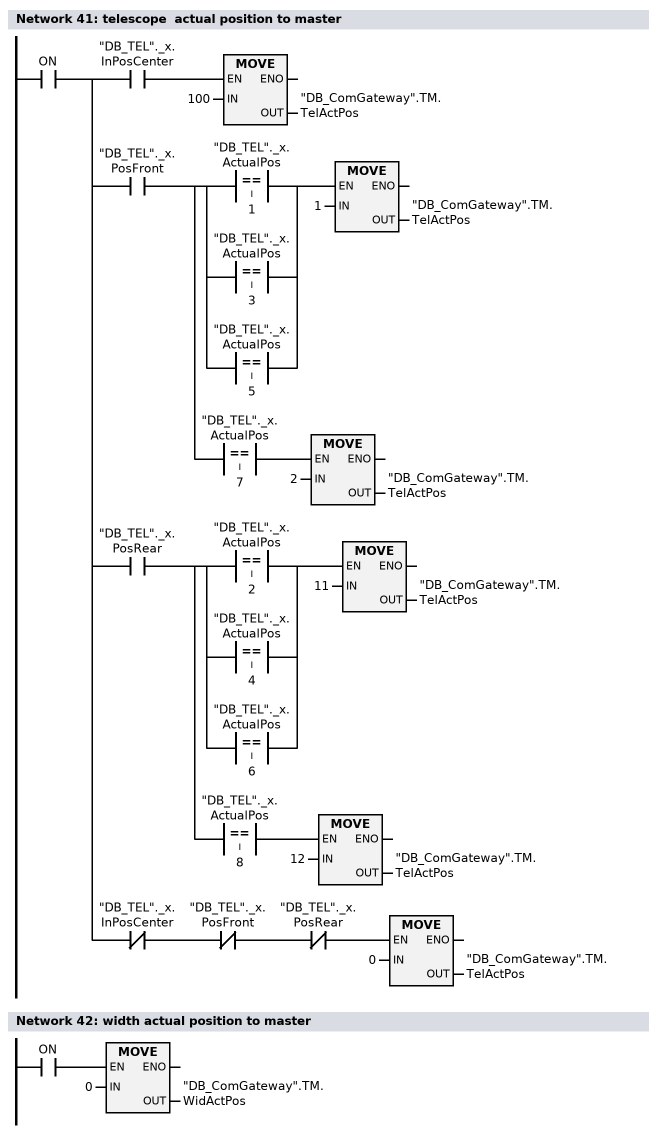
NETWORK
TITLE = telescope  actual position to master
      A     "ON";
      =     L 8.0;
      A     L 8.0;
      A     "DB_TEL"._x.InPosCenter;
      JNB   _02f;
      L     100;
      T     "DB_ComGateway".TM.TelActPos;
_02f: NOP   0;
      A     L 8.0;
      A     "DB_TEL"._x.PosFront;
      =     L 8.1;
      A     L 8.1;
      A(;
      O(;
      L     "DB_TEL"._x.ActualPos;
      L     1;
      ==I;
      );
      O(;
      L     "DB_TEL"._x.ActualPos;
      L     3;
      ==I;
      );
      O(;
      L     "DB_TEL"._x.ActualPos;
      L     5;
      ==I;
      );
      );
      JNB   _030;
      L     1;
      T     "DB_ComGateway".TM.TelActPos;
_030: NOP   0;
      A     L 8.1;
      A(;
      L     "DB_TEL"._x.ActualPos;
      L     7;
      ==I;
      );
      JNB   _031;
      L     2;
      T     "DB_ComGateway".TM.TelActPos;
_031: NOP   0;
      A     L 8.0;
      A     "DB_TEL"._x.PosRear;
      =     L 8.1;
      A     L 8.1;
      A(;
      O(;
      L     "DB_TEL"._x.ActualPos;
      L     2;
      ==I;
      );
      O(;
      L     "DB_TEL"._x.ActualPos;
      L     4;
      ==I;
      );
      O(;
      L     "DB_TEL"._x.ActualPos;
      L     6;
      ==I;
      );
      );
      JNB   _032;
      L     11;
      T     "DB_ComGateway".TM.TelActPos;
_032: NOP   0;
      A     L 8.1;
      A(;
      L     "DB_TEL"._x.ActualPos;
      L     8;
      ==I;
      );
      JNB   _033;
      L     12;
      T     "DB_ComGateway".TM.TelActPos;
_033: NOP   0;
      A     L 8.0;
      AN    "DB_TEL"._x.InPosCenter;
      AN    "DB_TEL"._x.PosFront;
      AN    "DB_TEL"._x.PosRear;
      JNB   _034;
      L     0;
      T     "DB_ComGateway".TM.TelActPos;
_034: NOP   0;
NETWORK
TITLE = width actual position to master
      A     "ON";
      JNB   _035;
      L     0;
      T     "DB_ComGateway".TM.WidActPos;
_035: NOP   0;
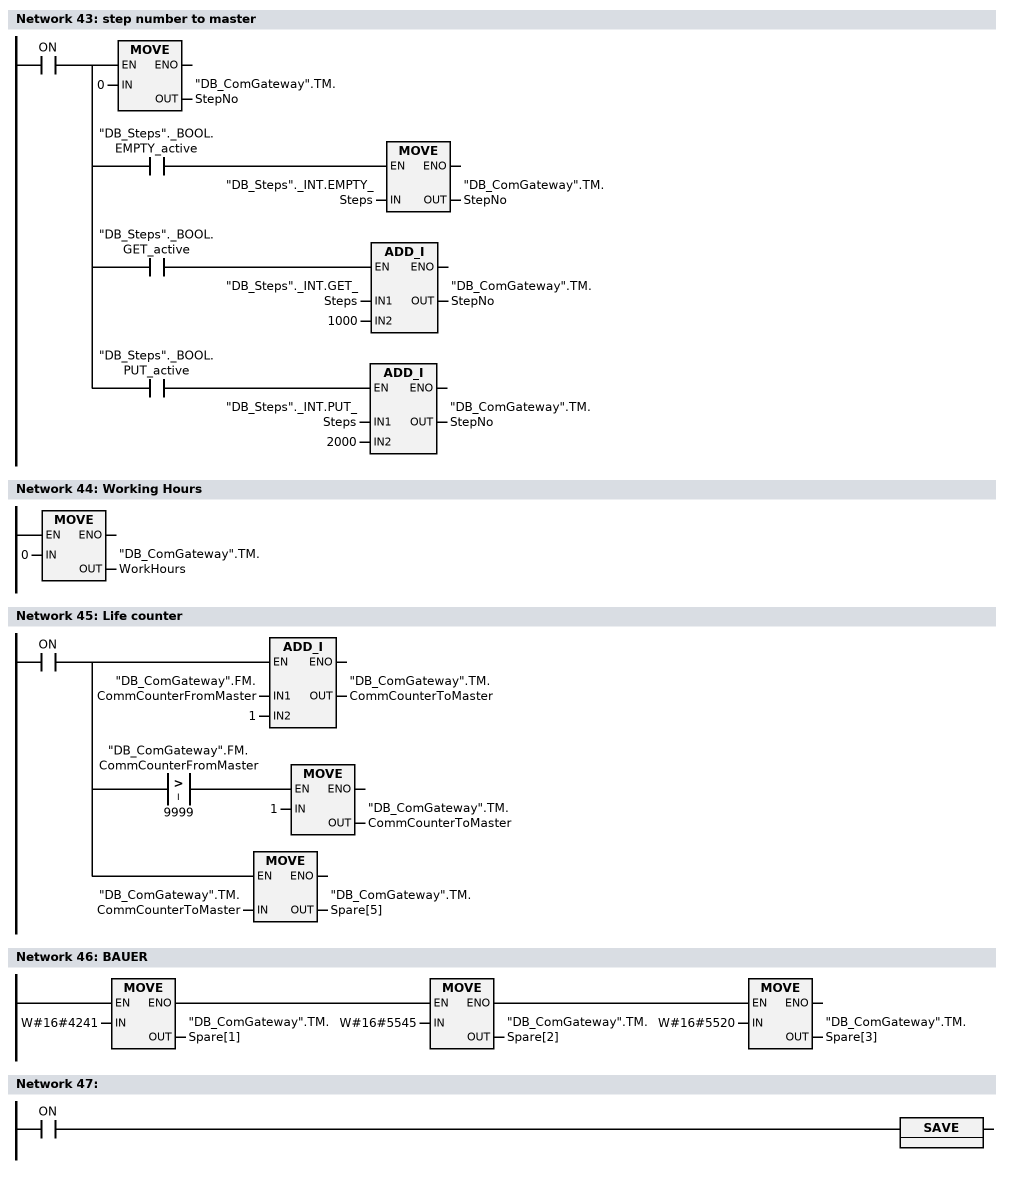
NETWORK
TITLE = step number to master
      A     "ON";
      =     L 8.0;
      A     L 8.0;
      JNB   _036;
      L     0;
      T     "DB_ComGateway".TM.StepNo;
_036: NOP   0;
      A     L 8.0;
      A     "DB_Steps"._BOOL.EMPTY_active;
      JNB   _037;
      L     "DB_Steps"._INT.EMPTY_Steps;
      T     "DB_ComGateway".TM.StepNo;
_037: NOP   0;
      A     L 8.0;
      A     "DB_Steps"._BOOL.GET_active;
      JNB   _038;
      L     "DB_Steps"._INT.GET_Steps;
      L     1000;
      +I;
      T     "DB_ComGateway".TM.StepNo;
_038: NOP   0;
      A     L 8.0;
      A     "DB_Steps"._BOOL.PUT_active;
      JNB   _039;
      L     "DB_Steps"._INT.PUT_Steps;
      L     2000;
      +I;
      T     "DB_ComGateway".TM.StepNo;
_039: NOP   0;
NETWORK
TITLE = Working Hours
      L     0;
      T     "DB_ComGateway".TM.WorkHours;
      NOP   0;
NETWORK
TITLE = Life counter
      A     "ON";
      =     L 8.0;
      A     L 8.0;
      JNB   _03a;
      L     "DB_ComGateway".FM.CommCounterFromMaster;
      L     1;
      +I;
      T     "DB_ComGateway".TM.CommCounterToMaster;
_03a: NOP   0;
      A     L 8.0;
      A(;
      L     "DB_ComGateway".FM.CommCounterFromMaster;
      L     9999;
      >I;
      );
      JNB   _03b;
      L     1;
      T     "DB_ComGateway".TM.CommCounterToMaster;
_03b: NOP   0;
      A     L 8.0;
      JNB   _03c;
      L     "DB_ComGateway".TM.CommCounterToMaster;
      T     "DB_ComGateway".TM.Spare[5];
_03c: NOP   0;
NETWORK
TITLE = BAUER
      A(;
      A(;
      L     W#16#4241;
      T     "DB_ComGateway".TM.Spare[1];
      SET;
      SAVE;
      CLR;
      A     BR;
      );
      JNB   _03d;
      L     W#16#5545;
      T     "DB_ComGateway".TM.Spare[2];
      SET;
      SAVE;
      CLR;
_03d: A     BR;
      );
      JNB   _03e;
      L     W#16#5520;
      T     "DB_ComGateway".TM.Spare[3];
_03e: NOP   0;
NETWORK
TITLE =
      A     "ON";
      SAVE;
END_FUNCTION

FUNCTION "STEPS_Control" : VOID	// FC 110
TITLE = Step Sequences
VERSION : 0.1
VAR_TEMP
  next : BOOL ;
  tmp_ActCircum : DINT ;
  tmp_CircumDiff : DINT ;
  tmp_OrderCircum : DINT ;
END_VAR
BEGIN
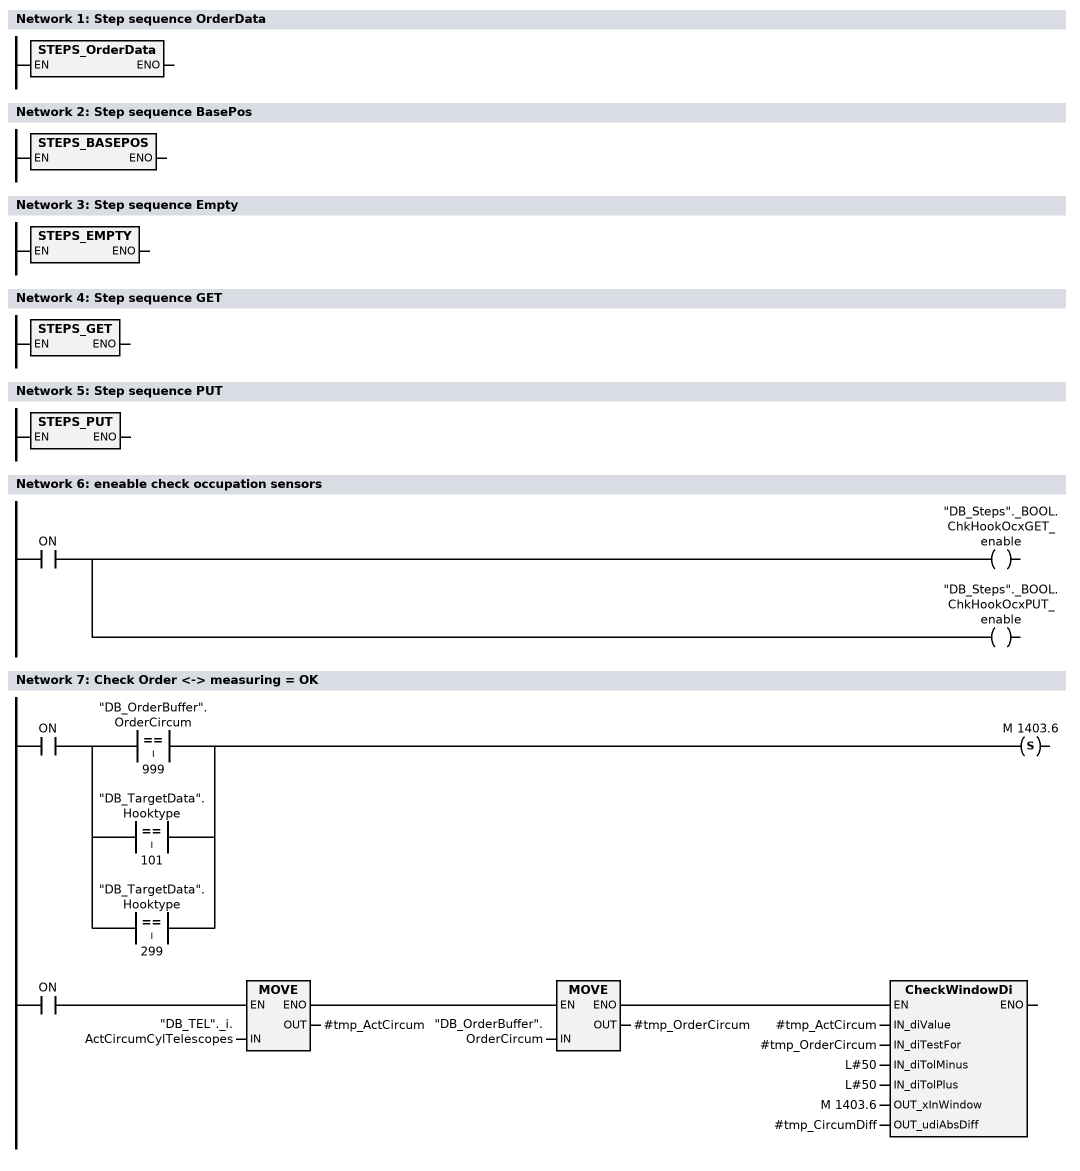
NETWORK
TITLE = Step sequence OrderData
      CALL  "STEPS_OrderData";
      NOP   0;
NETWORK
TITLE = Step sequence BasePos
      CALL  "STEPS_BASEPOS";
      NOP   0;
NETWORK
TITLE = Step sequence Empty
      CALL  "STEPS_EMPTY";
      NOP   0;
NETWORK
TITLE = Step sequence GET
      CALL  "STEPS_GET";
      NOP   0;
NETWORK
TITLE = Step sequence PUT
      CALL  "STEPS_PUT";
      NOP   0;
NETWORK
TITLE = eneable check occupation sensors
      A     "ON";
      =     "DB_Steps"._BOOL.ChkHookOcxGET_enable;
      =     "DB_Steps"._BOOL.ChkHookOcxPUT_enable;
NETWORK
TITLE = Check Order <-> measuring = OK
      A     "ON";
      =     L 14.0;
      A(;
      A(;
      A     L 14.0;
      JNB   _001;
      L     "DB_TEL"._i.ActCircumCylTelescopes;
      T     #tmp_ActCircum;
      SET;
      SAVE;
      CLR;
_001: A     BR;
      );
      JNB   _002;
      L     "DB_OrderBuffer".OrderCircum;
      T     #tmp_OrderCircum;
      SET;
      SAVE;
      CLR;
_002: A     BR;
      );
      JNB   _003;
      CALL  "CheckWindowDi" (
           IN_diValue               := #tmp_ActCircum,
           IN_diTestFor             := #tmp_OrderCircum,
           IN_diTolMinus            := L#50,
           IN_diTolPlus             := L#50,
           OUT_xInWindow            := M 1403.6,
           OUT_udiAbsDiff           := #tmp_CircumDiff);
_003: NOP   0;
      A     L 14.0;
      A(;
      O(;
      L     "DB_OrderBuffer".OrderCircum;
      L     999;
      ==I;
      );
      O(;
      L     "DB_TargetData".Hooktype;
      L     101;
      ==I;
      );
      O(;
      L     "DB_TargetData".Hooktype;
      L     299;
      ==I;
      );
      );
      S     M 1403.6;
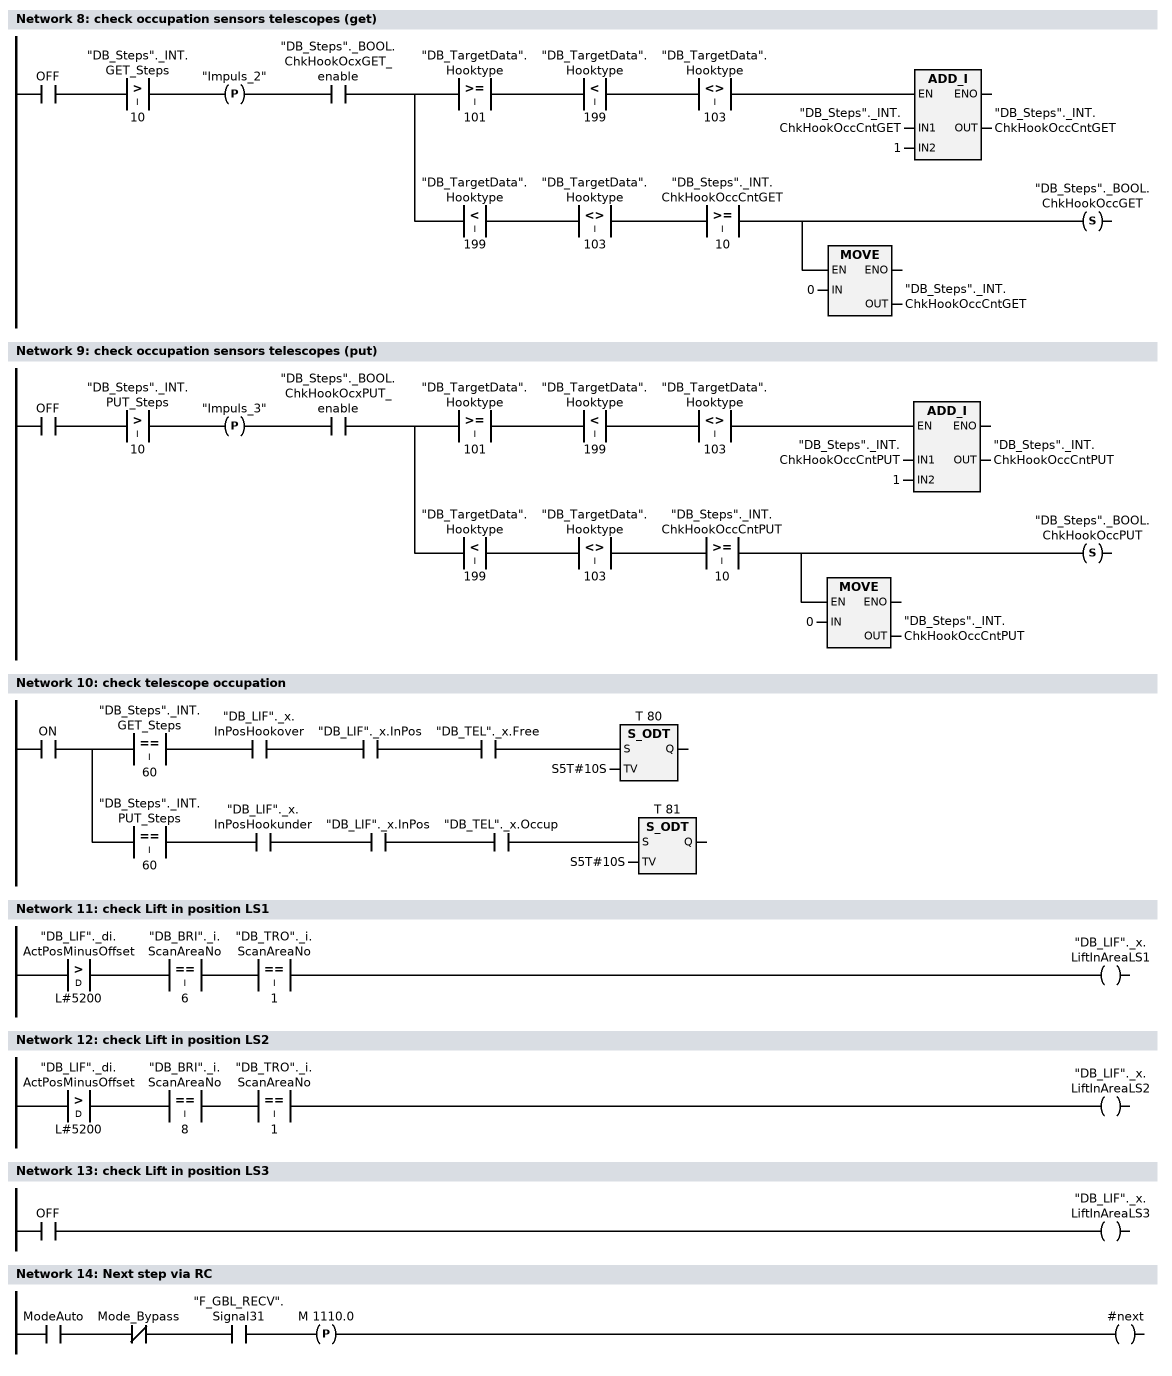
NETWORK
TITLE = check occupation sensors telescopes (get)
      A     "OFF";
      A(;
      L     "DB_Steps"._INT.GET_Steps;
      L     10;
      >I;
      );
      FP    "Impuls_2";
      A     "DB_Steps"._BOOL.ChkHookOcxGET_enable;
      =     L 14.0;
      A     L 14.0;
      A(;
      L     "DB_TargetData".Hooktype;
      L     101;
      >=I;
      );
      A(;
      L     "DB_TargetData".Hooktype;
      L     199;
      <I;
      );
      A(;
      L     "DB_TargetData".Hooktype;
      L     103;
      <>I;
      );
      JNB   _004;
      L     "DB_Steps"._INT.ChkHookOccCntGET;
      L     1;
      +I;
      T     "DB_Steps"._INT.ChkHookOccCntGET;
_004: NOP   0;
      A     L 14.0;
      A(;
      L     "DB_TargetData".Hooktype;
      L     199;
      <I;
      );
      A(;
      L     "DB_TargetData".Hooktype;
      L     103;
      <>I;
      );
      A(;
      L     "DB_Steps"._INT.ChkHookOccCntGET;
      L     10;
      >=I;
      );
      =     L 14.1;
      A     L 14.1;
      BLD   102;
      S     "DB_Steps"._BOOL.ChkHookOccGET;
      A     L 14.1;
      JNB   _005;
      L     0;
      T     "DB_Steps"._INT.ChkHookOccCntGET;
_005: NOP   0;
NETWORK
TITLE = check occupation sensors telescopes (put)
      A     "OFF";
      A(;
      L     "DB_Steps"._INT.PUT_Steps;
      L     10;
      >I;
      );
      FP    "Impuls_3";
      A     "DB_Steps"._BOOL.ChkHookOcxPUT_enable;
      =     L 14.0;
      A     L 14.0;
      A(;
      L     "DB_TargetData".Hooktype;
      L     101;
      >=I;
      );
      A(;
      L     "DB_TargetData".Hooktype;
      L     199;
      <I;
      );
      A(;
      L     "DB_TargetData".Hooktype;
      L     103;
      <>I;
      );
      JNB   _006;
      L     "DB_Steps"._INT.ChkHookOccCntPUT;
      L     1;
      +I;
      T     "DB_Steps"._INT.ChkHookOccCntPUT;
_006: NOP   0;
      A     L 14.0;
      A(;
      L     "DB_TargetData".Hooktype;
      L     199;
      <I;
      );
      A(;
      L     "DB_TargetData".Hooktype;
      L     103;
      <>I;
      );
      A(;
      L     "DB_Steps"._INT.ChkHookOccCntPUT;
      L     10;
      >=I;
      );
      =     L 14.1;
      A     L 14.1;
      BLD   102;
      S     "DB_Steps"._BOOL.ChkHookOccPUT;
      A     L 14.1;
      JNB   _007;
      L     0;
      T     "DB_Steps"._INT.ChkHookOccCntPUT;
_007: NOP   0;
NETWORK
TITLE = check telescope occupation
      A     "ON";
      =     L 14.0;
      A     L 14.0;
      A(;
      L     "DB_Steps"._INT.GET_Steps;
      L     60;
      ==I;
      );
      A     "DB_LIF"._x.InPosHookover;
      A     "DB_LIF"._x.InPos;
      A     "DB_TEL"._x.Free;
      L     S5T#10S;
      SD    T 80;
      NOP   0;
      NOP   0;
      NOP   0;
      NOP   0;
      A     L 14.0;
      A(;
      L     "DB_Steps"._INT.PUT_Steps;
      L     60;
      ==I;
      );
      A     "DB_LIF"._x.InPosHookunder;
      A     "DB_LIF"._x.InPos;
      A     "DB_TEL"._x.Occup;
      L     S5T#10S;
      SD    T 81;
      NOP   0;
      NOP   0;
      NOP   0;
      NOP   0;
NETWORK
TITLE = check Lift in position LS1
      A(;
      L     "DB_LIF"._di.ActPosMinusOffset;
      L     L#5200;
      >D;
      );
      A(;
      L     "DB_BRI"._i.ScanAreaNo;
      L     6;
      ==I;
      );
      A(;
      L     "DB_TRO"._i.ScanAreaNo;
      L     1;
      ==I;
      );
      =     "DB_LIF"._x.LiftInAreaLS1;
NETWORK
TITLE = check Lift in position LS2
      A(;
      L     "DB_LIF"._di.ActPosMinusOffset;
      L     L#5200;
      >D;
      );
      A(;
      L     "DB_BRI"._i.ScanAreaNo;
      L     8;
      ==I;
      );
      A(;
      L     "DB_TRO"._i.ScanAreaNo;
      L     1;
      ==I;
      );
      =     "DB_LIF"._x.LiftInAreaLS2;
NETWORK
TITLE = check Lift in position LS3
      A     "OFF";
      =     "DB_LIF"._x.LiftInAreaLS3;
NETWORK
TITLE = Next step via RC
      A     "ModeAuto";
      AN    "Mode_Bypass";
      A     "F_GBL_RECV".Signal31;
      FP    M 1110.0;
      =     #next;
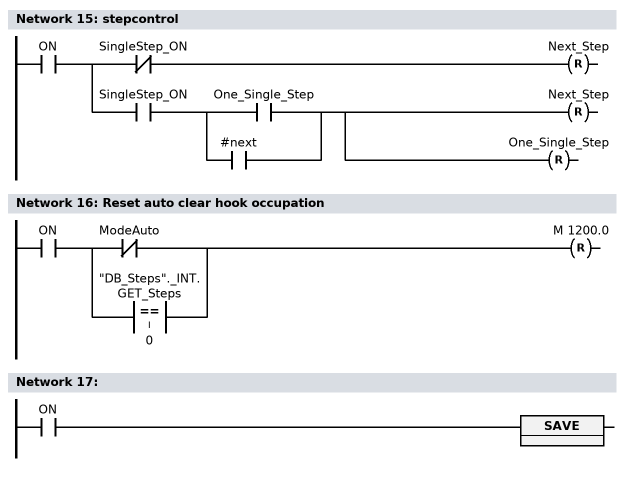
NETWORK
TITLE = stepcontrol
//Einzelschritt
      A     "ON";
      =     L 14.0;
      A     L 14.0;
      AN    "SingleStep_ON";
      R     "Next_Step";
      A     L 14.0;
      A     "SingleStep_ON";
      A(;
      O     "One_Single_Step";
      O     #next;
      );
      R     "Next_Step";
      R     "One_Single_Step";
NETWORK
TITLE = Reset auto clear hook occupation
      A     "ON";
      A(;
      ON    "ModeAuto";
      O(;
      L     "DB_Steps"._INT.GET_Steps;
      L     0;
      ==I;
      );
      );
      R     M 1200.0;
NETWORK
TITLE =
      A     "ON";
      SAVE;
END_FUNCTION

FUNCTION "STEPS_OrderData" : VOID	// FC 111
TITLE = Steps OrderData
VERSION : 2.0
VAR_TEMP
  tmp_OrderPosValBRI : DINT ;
  tmp_di_1 : DINT ;
  tmp_di_DiffHoHu : DINT ;
  tmp_RetValErrCode : INT ;
  tmp_LifTargetPosNo : INT ;
  tmp_RetValErrCodeBRI : INT ;
  tmp_OrderPosNoBRI : INT ;
  tmp_OrderLIF_DBNo : INT ;
  tmp_OrderLIF_DBNo_2 : INT ;
  tmp_RetValErrBRI : BOOL ;
  tmp_TRO_DataOk : BOOL ;
  tmp_LIF_DataOK : BOOL ;
  tmp_TEL_DataOK : BOOL ;
  tmp_LifReleaseTarg : BOOL ;
  tmp_BriDataOK : BOOL ;
  tmp_LifTargetDataOK : BOOL ;
  tmp_OrderPosNoTRO : INT ;
  tmp_OrderPosValTRO : DINT ;
  tmp_TRBR : INT ;
  tmp_WID_DataOK : BOOL ;
  tmp_ReadDB_OK : BOOL ;
  tmp_StartDBCopy : BOOL ;
END_VAR
BEGIN
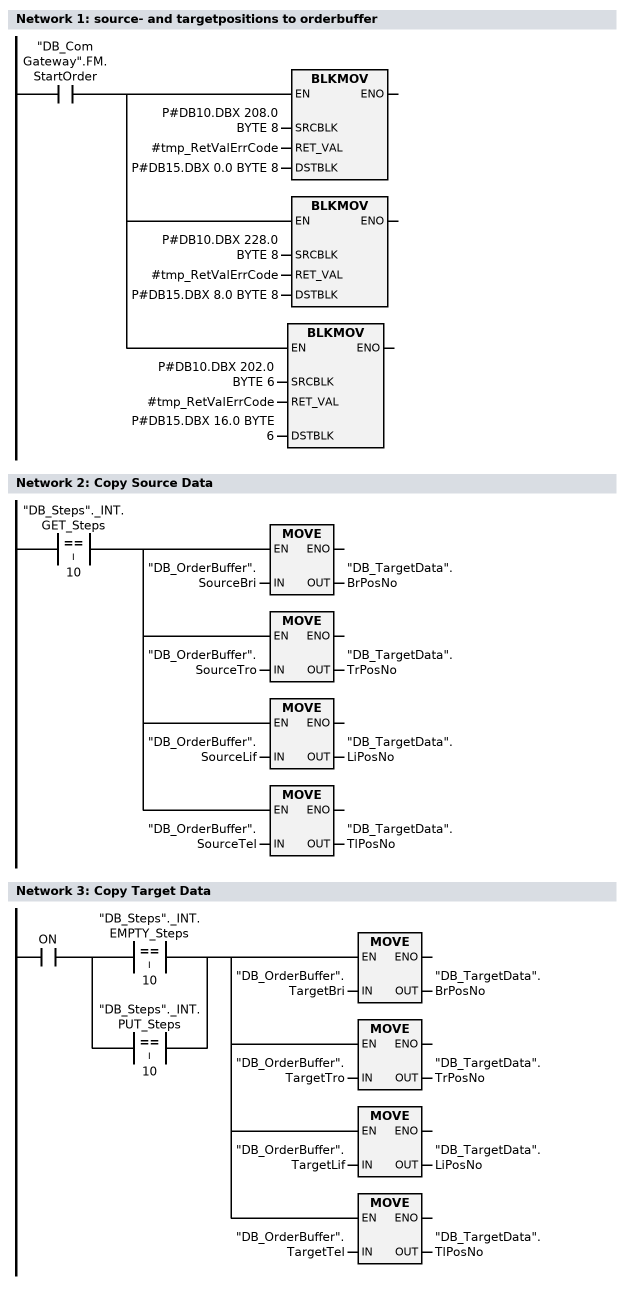
NETWORK
TITLE = source- and targetpositions to orderbuffer
      A     "DB_ComGateway".FM.StartOrder;
      =     L 35.0;
      A     L 35.0;
      JNB   _001;
      CALL  "BLKMOV" (
           SRCBLK                   := P#DB10.DBX 208.0 BYTE 8,
           RET_VAL                  := #tmp_RetValErrCode,
           DSTBLK                   := P#DB15.DBX 0.0 BYTE 8);
_001: NOP   0;
      A     L 35.0;
      JNB   _002;
      CALL  "BLKMOV" (
           SRCBLK                   := P#DB10.DBX 228.0 BYTE 8,
           RET_VAL                  := #tmp_RetValErrCode,
           DSTBLK                   := P#DB15.DBX 8.0 BYTE 8);
_002: NOP   0;
      A     L 35.0;
      JNB   _003;
      CALL  "BLKMOV" (
           SRCBLK                   := P#DB10.DBX 202.0 BYTE 6,
           RET_VAL                  := #tmp_RetValErrCode,
           DSTBLK                   := P#DB15.DBX 16.0 BYTE 6);
_003: NOP   0;
NETWORK
TITLE = Copy Source Data
      L     "DB_Steps"._INT.GET_Steps;
      L     10;
      ==I;
      =     L 35.0;
      A     L 35.0;
      JNB   _004;
      L     "DB_OrderBuffer".SourceBri;
      T     "DB_TargetData".BrPosNo;
_004: NOP   0;
      A     L 35.0;
      JNB   _005;
      L     "DB_OrderBuffer".SourceTro;
      T     "DB_TargetData".TrPosNo;
_005: NOP   0;
      A     L 35.0;
      JNB   _006;
      L     "DB_OrderBuffer".SourceLif;
      T     "DB_TargetData".LiPosNo;
_006: NOP   0;
      A     L 35.0;
      JNB   _007;
      L     "DB_OrderBuffer".SourceTel;
      T     "DB_TargetData".TlPosNo;
_007: NOP   0;
NETWORK
TITLE = Copy Target Data
      A     "ON";
      A(;
      O(;
      L     "DB_Steps"._INT.EMPTY_Steps;
      L     10;
      ==I;
      );
      O(;
      L     "DB_Steps"._INT.PUT_Steps;
      L     10;
      ==I;
      );
      );
      =     L 35.0;
      A     L 35.0;
      JNB   _008;
      L     "DB_OrderBuffer".TargetBri;
      T     "DB_TargetData".BrPosNo;
_008: NOP   0;
      A     L 35.0;
      JNB   _009;
      L     "DB_OrderBuffer".TargetTro;
      T     "DB_TargetData".TrPosNo;
_009: NOP   0;
      A     L 35.0;
      JNB   _00a;
      L     "DB_OrderBuffer".TargetLif;
      T     "DB_TargetData".LiPosNo;
_00a: NOP   0;
      A     L 35.0;
      JNB   _00b;
      L     "DB_OrderBuffer".TargetTel;
      T     "DB_TargetData".TlPosNo;
_00b: NOP   0;
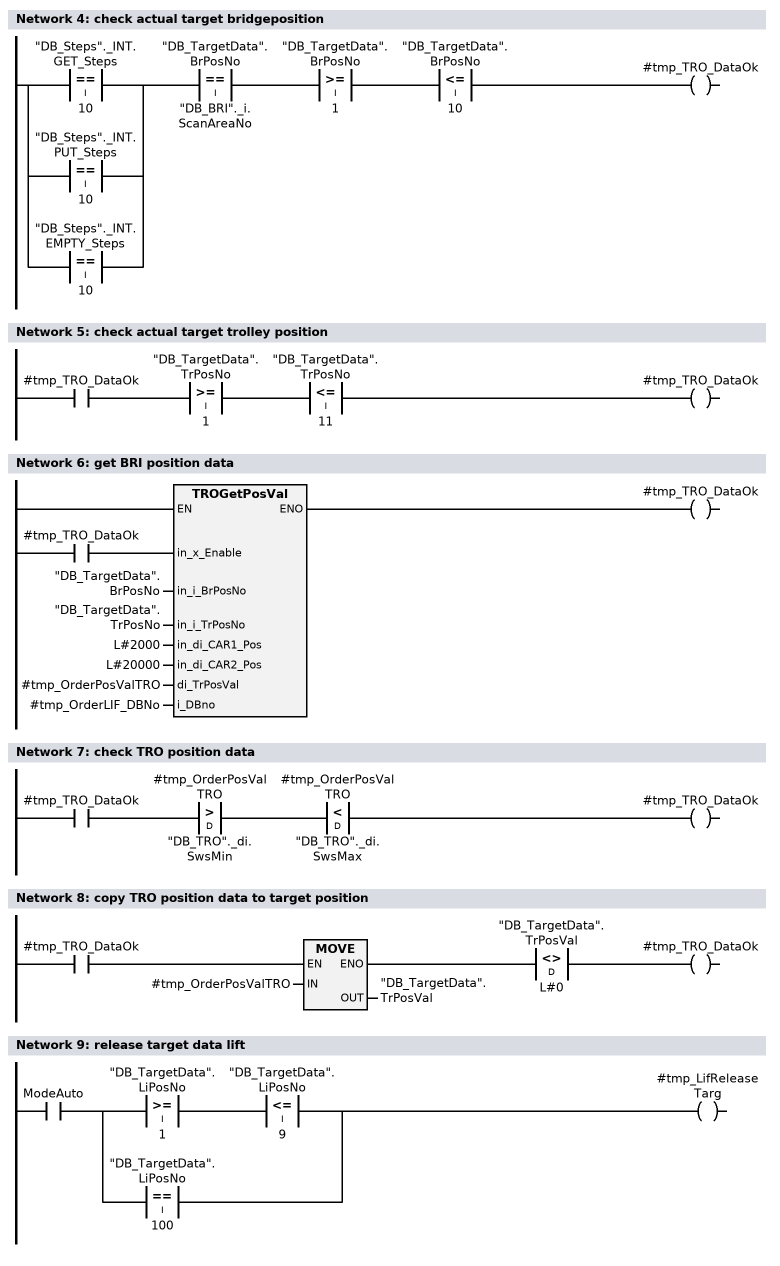
NETWORK
TITLE = check actual target bridgeposition
//because the RBG MUST in same tower we allow only if order is same too
      A(;
      O(;
      L     "DB_Steps"._INT.GET_Steps;
      L     10;
      ==I;
      );
      O(;
      L     "DB_Steps"._INT.PUT_Steps;
      L     10;
      ==I;
      );
      O(;
      L     "DB_Steps"._INT.EMPTY_Steps;
      L     10;
      ==I;
      );
      );
      A(;
      L     "DB_TargetData".BrPosNo;
      L     "DB_BRI"._i.ScanAreaNo;
      ==I;
      );
      A(;
      L     "DB_TargetData".BrPosNo;
      L     1;
      >=I;
      );
      A(;
      L     "DB_TargetData".BrPosNo;
      L     10;
      <=I;
      );
      =     #tmp_TRO_DataOk;
NETWORK
TITLE = check actual target trolley position 
      A     #tmp_TRO_DataOk;
      A(;
      L     "DB_TargetData".TrPosNo;
      L     1;
      >=I;
      );
      A(;
      L     "DB_TargetData".TrPosNo;
      L     11;
      <=I;
      );
      =     #tmp_TRO_DataOk;
NETWORK
TITLE = get BRI position data
//TODO values carrier 1/2
      A     #tmp_TRO_DataOk;
      =     L 35.0;
      BLD   103;
      CALL  "TROGetPosVal" (
           in_x_Enable              := L 35.0,
           in_i_BrPosNo             := "DB_TargetData".BrPosNo,
           in_i_TrPosNo             := "DB_TargetData".TrPosNo,
           in_di_CAR1_Pos           := L#2000,
           in_di_CAR2_Pos           := L#20000,
           di_TrPosVal              := #tmp_OrderPosValTRO,
           i_DBno                   := #tmp_OrderLIF_DBNo);
      A     BR;
      =     #tmp_TRO_DataOk;
NETWORK
TITLE = check TRO position data
      A     #tmp_TRO_DataOk;
      A(;
      L     #tmp_OrderPosValTRO;
      L     "DB_TRO"._di.SwsMin;
      >D;
      );
      A(;
      L     #tmp_OrderPosValTRO;
      L     "DB_TRO"._di.SwsMax;
      <D;
      );
      =     #tmp_TRO_DataOk;
NETWORK
TITLE = copy TRO position data to target position
      A(;
      A     #tmp_TRO_DataOk;
      JNB   _00c;
      L     #tmp_OrderPosValTRO;
      T     "DB_TargetData".TrPosVal;
      SET;
      SAVE;
      CLR;
_00c: A     BR;
      );
      A(;
      L     "DB_TargetData".TrPosVal;
      L     L#0;
      <>D;
      );
      =     #tmp_TRO_DataOk;
NETWORK
TITLE = release target data lift
      A     "ModeAuto";
      A(;
      A(;
      L     "DB_TargetData".LiPosNo;
      L     1;
      >=I;
      );
      A(;
      L     "DB_TargetData".LiPosNo;
      L     9;
      <=I;
      );
      O(;
      L     "DB_TargetData".LiPosNo;
      L     100;
      ==I;
      );
      );
      =     #tmp_LifReleaseTarg;
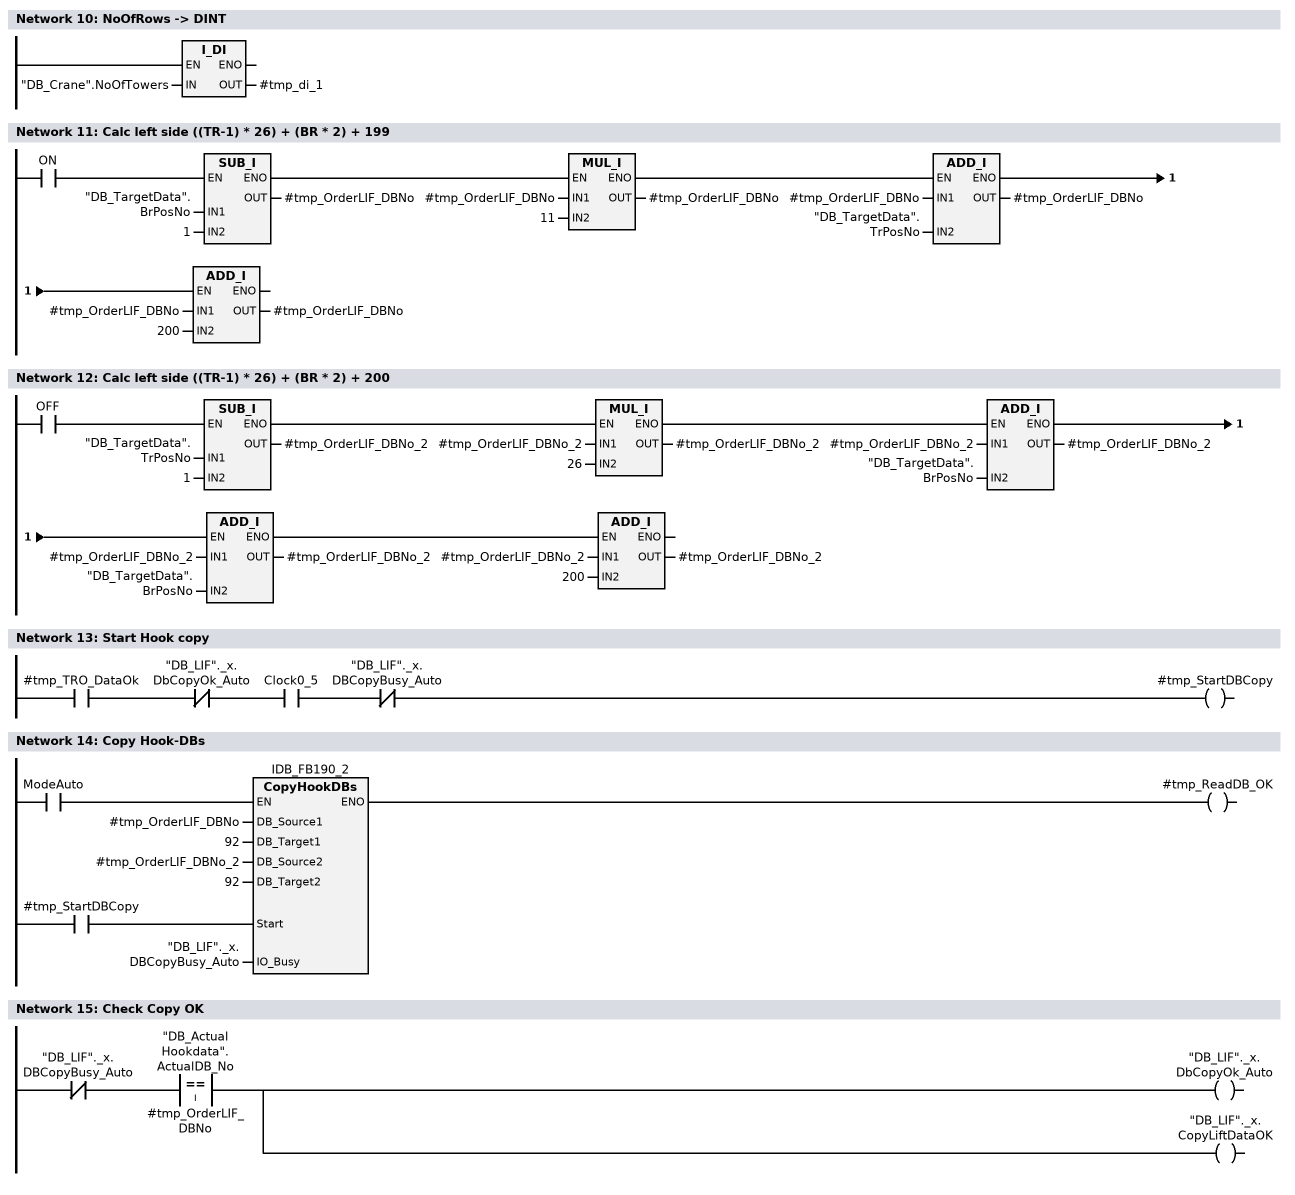
NETWORK
TITLE = NoOfRows -> DINT
      L     "DB_Crane".NoOfTowers;
      ITD;
      T     #tmp_di_1;
      NOP   0;
NETWORK
TITLE = Calc left side ((TR-1) * 26) + (BR * 2) + 199
      A(;
      A(;
      A(;
      A     "ON";
      JNB   _00d;
      L     "DB_TargetData".BrPosNo;
      L     1;
      -I;
      T     #tmp_OrderLIF_DBNo;
      AN    OV;
      SAVE;
      CLR;
_00d: A     BR;
      );
      JNB   _00e;
      L     #tmp_OrderLIF_DBNo;
      L     11;
      *I;
      T     #tmp_OrderLIF_DBNo;
      AN    OV;
      SAVE;
      CLR;
_00e: A     BR;
      );
      JNB   _00f;
      L     #tmp_OrderLIF_DBNo;
      L     "DB_TargetData".TrPosNo;
      +I;
      T     #tmp_OrderLIF_DBNo;
      AN    OV;
      SAVE;
      CLR;
_00f: A     BR;
      );
      JNB   _010;
      L     #tmp_OrderLIF_DBNo;
      L     200;
      +I;
      T     #tmp_OrderLIF_DBNo;
_010: NOP   0;
NETWORK
TITLE = Calc left side ((TR-1) * 26) + (BR * 2) + 200
      A(;
      A(;
      A(;
      A(;
      A     "OFF";
      JNB   _011;
      L     "DB_TargetData".TrPosNo;
      L     1;
      -I;
      T     #tmp_OrderLIF_DBNo_2;
      AN    OV;
      SAVE;
      CLR;
_011: A     BR;
      );
      JNB   _012;
      L     #tmp_OrderLIF_DBNo_2;
      L     26;
      *I;
      T     #tmp_OrderLIF_DBNo_2;
      AN    OV;
      SAVE;
      CLR;
_012: A     BR;
      );
      JNB   _013;
      L     #tmp_OrderLIF_DBNo_2;
      L     "DB_TargetData".BrPosNo;
      +I;
      T     #tmp_OrderLIF_DBNo_2;
      AN    OV;
      SAVE;
      CLR;
_013: A     BR;
      );
      JNB   _014;
      L     #tmp_OrderLIF_DBNo_2;
      L     "DB_TargetData".BrPosNo;
      +I;
      T     #tmp_OrderLIF_DBNo_2;
      AN    OV;
      SAVE;
      CLR;
_014: A     BR;
      );
      JNB   _015;
      L     #tmp_OrderLIF_DBNo_2;
      L     200;
      +I;
      T     #tmp_OrderLIF_DBNo_2;
_015: NOP   0;
NETWORK
TITLE = Start Hook copy
      A     #tmp_TRO_DataOk;
      AN    "DB_LIF"._x.DbCopyOk_Auto;
      A     "Clock0_5";
      AN    "DB_LIF"._x.DBCopyBusy_Auto;
      =     #tmp_StartDBCopy;
NETWORK
TITLE = Copy Hook-DBs
      A     #tmp_StartDBCopy;
      =     L 35.0;
      BLD   103;
      A     "ModeAuto";
      JNB   _016;
      CALL  "CopyHookDBs" , "IDB_FB190_2" (
           DB_Source1               := #tmp_OrderLIF_DBNo,
           DB_Target1               := 92,
           DB_Source2               := #tmp_OrderLIF_DBNo_2,
           DB_Target2               := 92,
           Start                    := L 35.0,
           IO_Busy                  := "DB_LIF"._x.DBCopyBusy_Auto);
_016: A     BR;
      =     #tmp_ReadDB_OK;
NETWORK
TITLE = Check Copy OK
      AN    "DB_LIF"._x.DBCopyBusy_Auto;
      A(;
      L     "DB_ActualHookdata".ActualDB_No;
      L     #tmp_OrderLIF_DBNo;
      ==I;
      );
      =     "DB_LIF"._x.DbCopyOk_Auto;
      =     "DB_LIF"._x.CopyLiftDataOK;
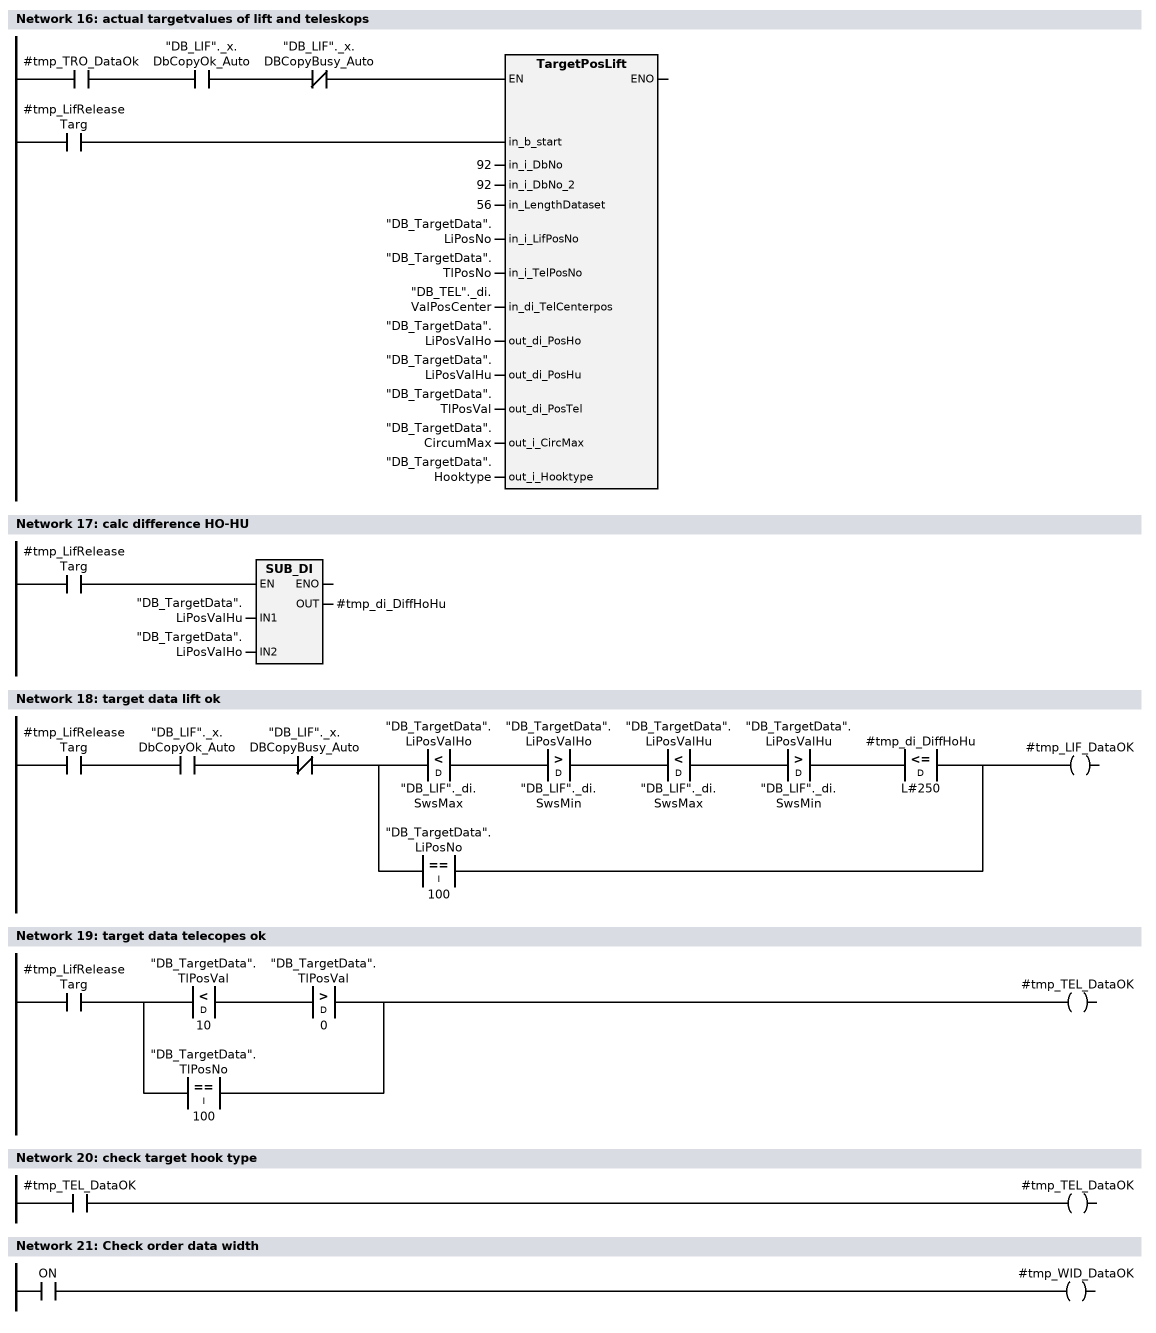
NETWORK
TITLE = actual targetvalues of lift and teleskops
      A     #tmp_LifReleaseTarg;
      =     L 35.0;
      BLD   103;
      A     #tmp_TRO_DataOk;
      A     "DB_LIF"._x.DbCopyOk_Auto;
      AN    "DB_LIF"._x.DBCopyBusy_Auto;
      JNB   _017;
      CALL  "TargetPosLift" (
           in_b_start               := L 35.0,
           in_i_DbNo                := 92,
           in_i_DbNo_2              := 92,
           in_LengthDataset         := 56,
           in_i_LifPosNo            := "DB_TargetData".LiPosNo,
           in_i_TelPosNo            := "DB_TargetData".TlPosNo,
           in_di_TelCenterpos       := "DB_TEL"._di.ValPosCenter,
           out_di_PosHo             := "DB_TargetData".LiPosValHo,
           out_di_PosHu             := "DB_TargetData".LiPosValHu,
           out_di_PosTel            := "DB_TargetData".TlPosVal,
           out_i_CircMax            := "DB_TargetData".CircumMax,
           out_i_Hooktype           := "DB_TargetData".Hooktype);
_017: NOP   0;
NETWORK
TITLE = calc difference HO-HU
      A     #tmp_LifReleaseTarg;
      JNB   _018;
      L     "DB_TargetData".LiPosValHu;
      L     "DB_TargetData".LiPosValHo;
      -D;
      T     #tmp_di_DiffHoHu;
_018: NOP   0;
NETWORK
TITLE = target data lift ok
      A     #tmp_LifReleaseTarg;
      A     "DB_LIF"._x.DbCopyOk_Auto;
      AN    "DB_LIF"._x.DBCopyBusy_Auto;
      A(;
      A(;
      L     "DB_TargetData".LiPosValHo;
      L     "DB_LIF"._di.SwsMax;
      <D;
      );
      A(;
      L     "DB_TargetData".LiPosValHo;
      L     "DB_LIF"._di.SwsMin;
      >D;
      );
      A(;
      L     "DB_TargetData".LiPosValHu;
      L     "DB_LIF"._di.SwsMax;
      <D;
      );
      A(;
      L     "DB_TargetData".LiPosValHu;
      L     "DB_LIF"._di.SwsMin;
      >D;
      );
      A(;
      L     #tmp_di_DiffHoHu;
      L     L#250;
      <=D;
      );
      O(;
      L     "DB_TargetData".LiPosNo;
      L     100;
      ==I;
      );
      );
      =     #tmp_LIF_DataOK;
NETWORK
TITLE = target data telecopes ok
      A     #tmp_LifReleaseTarg;
      A(;
      A(;
      L     "DB_TargetData".TlPosVal;
      L     10;
      <D;
      );
      A(;
      L     "DB_TargetData".TlPosVal;
      L     0;
      >D;
      );
      O(;
      L     "DB_TargetData".TlPosNo;
      L     100;
      ==I;
      );
      );
      =     #tmp_TEL_DataOK;
NETWORK
TITLE = check target hook type
      A     #tmp_TEL_DataOK;
      =     #tmp_TEL_DataOK;
NETWORK
TITLE = Check order data width
      A     "ON";
      =     #tmp_WID_DataOK;
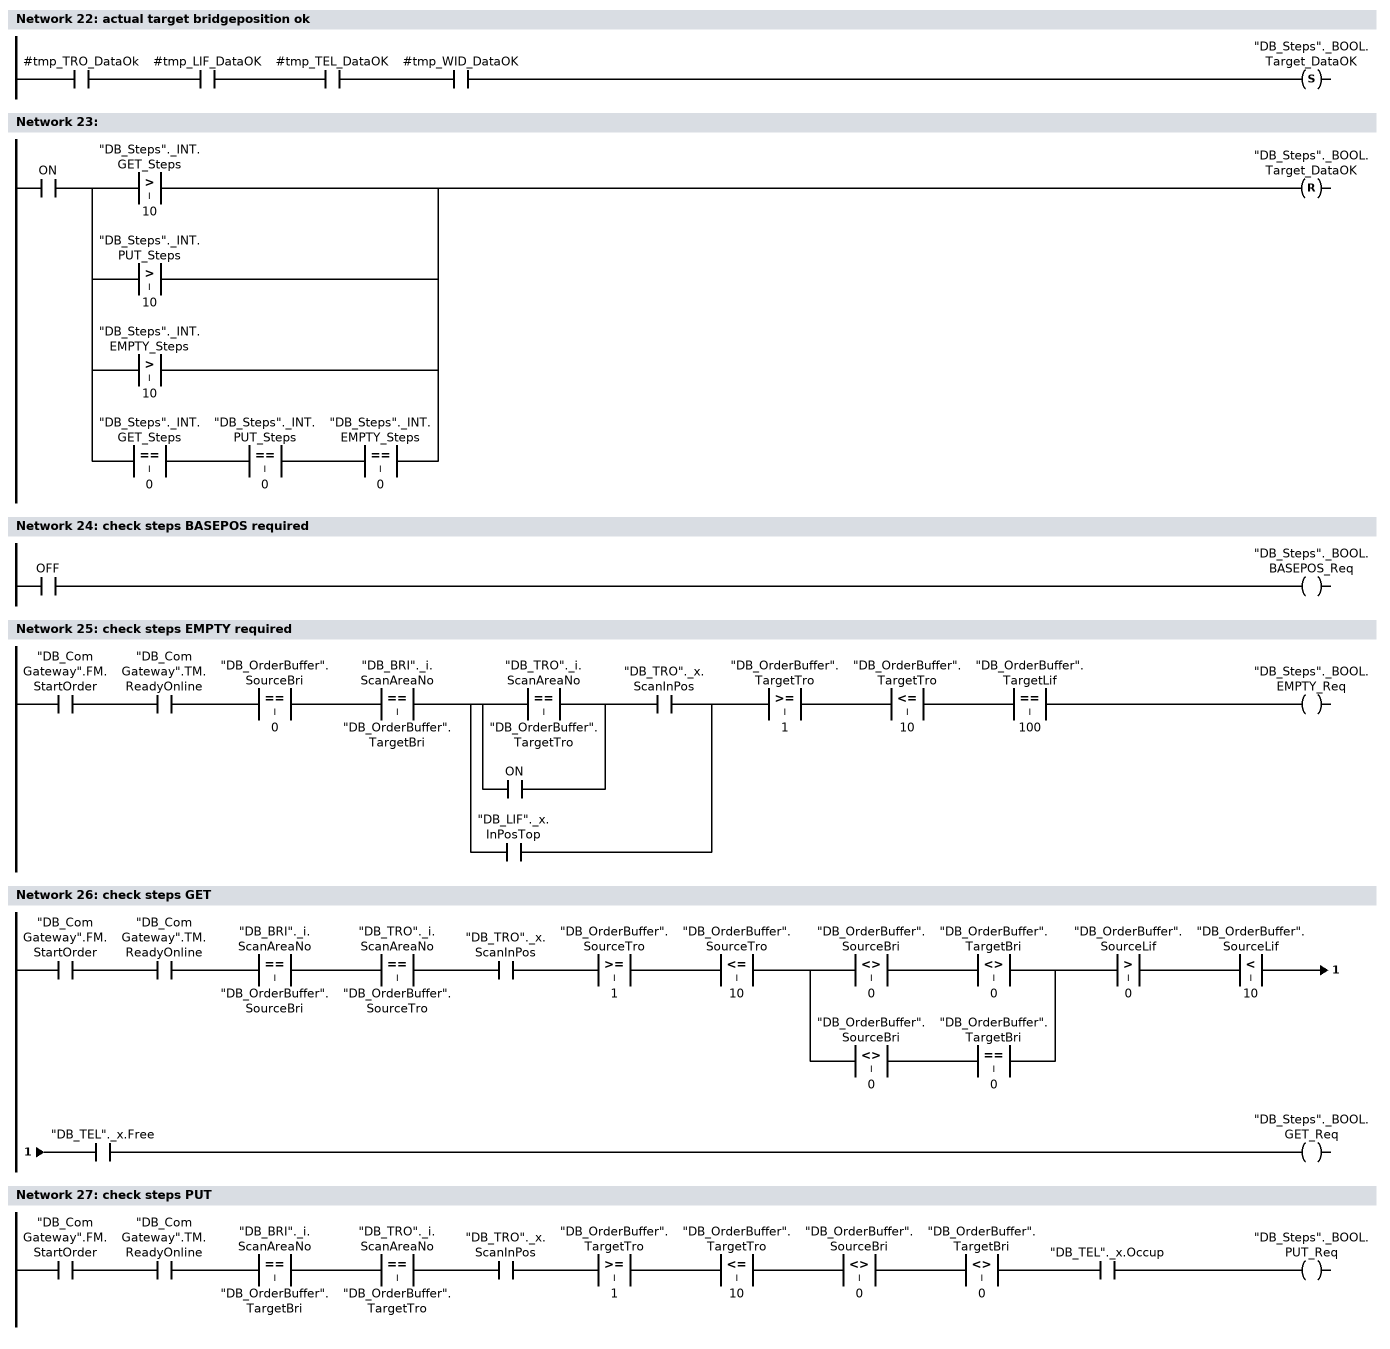
NETWORK
TITLE = actual target bridgeposition ok
      A     #tmp_TRO_DataOk;
      A     #tmp_LIF_DataOK;
      A     #tmp_TEL_DataOK;
      A     #tmp_WID_DataOK;
      S     "DB_Steps"._BOOL.Target_DataOK;
NETWORK
TITLE =
      A     "ON";
      A(;
      O(;
      L     "DB_Steps"._INT.GET_Steps;
      L     10;
      >I;
      );
      O(;
      L     "DB_Steps"._INT.PUT_Steps;
      L     10;
      >I;
      );
      O(;
      L     "DB_Steps"._INT.EMPTY_Steps;
      L     10;
      >I;
      );
      O;
      A(;
      L     "DB_Steps"._INT.GET_Steps;
      L     0;
      ==I;
      );
      A(;
      L     "DB_Steps"._INT.PUT_Steps;
      L     0;
      ==I;
      );
      A(;
      L     "DB_Steps"._INT.EMPTY_Steps;
      L     0;
      ==I;
      );
      );
      R     "DB_Steps"._BOOL.Target_DataOK;
NETWORK
TITLE = check steps BASEPOS required
      A     "OFF";
      =     "DB_Steps"._BOOL.BASEPOS_Req;
NETWORK
TITLE = check steps EMPTY required
//Source=0 and Target<>0
      A     "DB_ComGateway".FM.StartOrder;
      A     "DB_ComGateway".TM.ReadyOnline;
      A(;
      L     "DB_OrderBuffer".SourceBri;
      L     0;
      ==I;
      );
      A(;
      L     "DB_BRI"._i.ScanAreaNo;
      L     "DB_OrderBuffer".TargetBri;
      ==I;
      );
      A(;
      A(;
      O(;
      L     "DB_TRO"._i.ScanAreaNo;
      L     "DB_OrderBuffer".TargetTro;
      ==I;
      );
      O     "ON";
      );
      A     "DB_TRO"._x.ScanInPos;
      O     "DB_LIF"._x.InPosTop;
      );
      A(;
      L     "DB_OrderBuffer".TargetTro;
      L     1;
      >=I;
      );
      A(;
      L     "DB_OrderBuffer".TargetTro;
      L     10;
      <=I;
      );
      A(;
      L     "DB_OrderBuffer".TargetLif;
      L     100;
      ==I;
      );
      =     "DB_Steps"._BOOL.EMPTY_Req;
NETWORK
TITLE = check steps GET
//two possibilities:
// Source<>0 and Target=0
// Source<>0 and Target<>0
//not carrier
      A     "DB_ComGateway".FM.StartOrder;
      A     "DB_ComGateway".TM.ReadyOnline;
      A(;
      L     "DB_BRI"._i.ScanAreaNo;
      L     "DB_OrderBuffer".SourceBri;
      ==I;
      );
      A(;
      L     "DB_TRO"._i.ScanAreaNo;
      L     "DB_OrderBuffer".SourceTro;
      ==I;
      );
      A     "DB_TRO"._x.ScanInPos;
      A(;
      L     "DB_OrderBuffer".SourceTro;
      L     1;
      >=I;
      );
      A(;
      L     "DB_OrderBuffer".SourceTro;
      L     10;
      <=I;
      );
      A(;
      A(;
      L     "DB_OrderBuffer".SourceBri;
      L     0;
      <>I;
      );
      A(;
      L     "DB_OrderBuffer".TargetBri;
      L     0;
      <>I;
      );
      O;
      A(;
      L     "DB_OrderBuffer".SourceBri;
      L     0;
      <>I;
      );
      A(;
      L     "DB_OrderBuffer".TargetBri;
      L     0;
      ==I;
      );
      );
      A(;
      L     "DB_OrderBuffer".SourceLif;
      L     0;
      >I;
      );
      A(;
      L     "DB_OrderBuffer".SourceLif;
      L     10;
      <I;
      );
      A     "DB_TEL"._x.Free;
      =     "DB_Steps"._BOOL.GET_Req;
NETWORK
TITLE = check steps PUT
//Source<>0 and Target<>0 and occupied
//not carrier
      A     "DB_ComGateway".FM.StartOrder;
      A     "DB_ComGateway".TM.ReadyOnline;
      A(;
      L     "DB_BRI"._i.ScanAreaNo;
      L     "DB_OrderBuffer".TargetBri;
      ==I;
      );
      A(;
      L     "DB_TRO"._i.ScanAreaNo;
      L     "DB_OrderBuffer".TargetTro;
      ==I;
      );
      A     "DB_TRO"._x.ScanInPos;
      A(;
      L     "DB_OrderBuffer".TargetTro;
      L     1;
      >=I;
      );
      A(;
      L     "DB_OrderBuffer".TargetTro;
      L     10;
      <=I;
      );
      A(;
      L     "DB_OrderBuffer".SourceBri;
      L     0;
      <>I;
      );
      A(;
      L     "DB_OrderBuffer".TargetBri;
      L     0;
      <>I;
      );
      A     "DB_TEL"._x.Occup;
      =     "DB_Steps"._BOOL.PUT_Req;
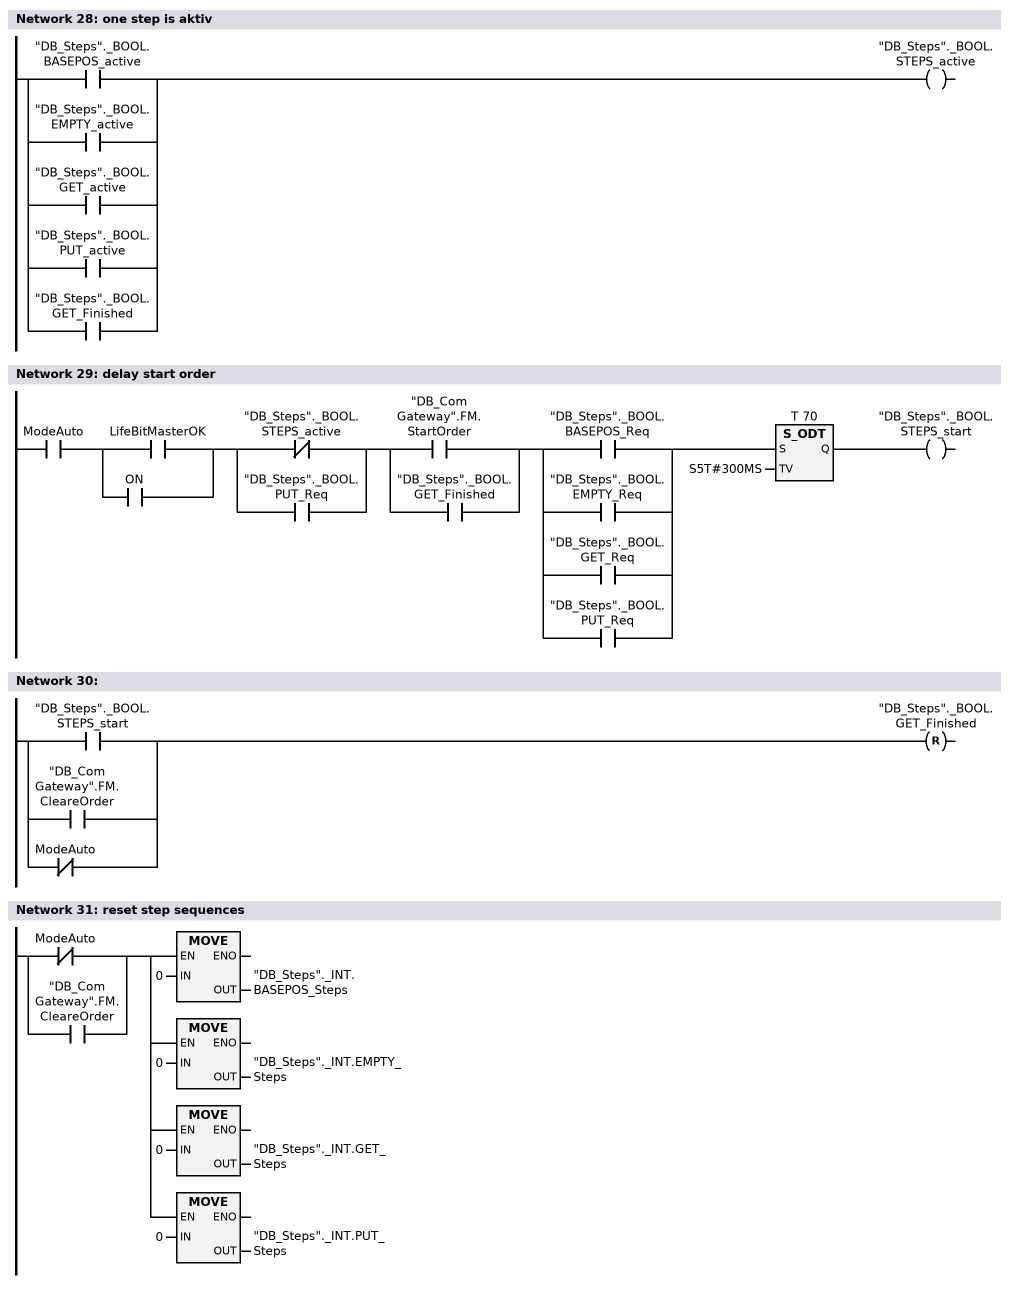
NETWORK
TITLE = one step is aktiv
      O     "DB_Steps"._BOOL.BASEPOS_active;
      O     "DB_Steps"._BOOL.EMPTY_active;
      O     "DB_Steps"._BOOL.GET_active;
      O     "DB_Steps"._BOOL.PUT_active;
      O     "DB_Steps"._BOOL.GET_Finished;
      =     "DB_Steps"._BOOL.STEPS_active;
NETWORK
TITLE = delay start order
      A     "ModeAuto";
      A(;
      O     "LifeBitMasterOK";
      O     "ON";
      );
      A(;
      ON    "DB_Steps"._BOOL.STEPS_active;
      O     "DB_Steps"._BOOL.PUT_Req;
      );
      A(;
      O     "DB_ComGateway".FM.StartOrder;
      O     "DB_Steps"._BOOL.GET_Finished;
      );
      A(;
      O     "DB_Steps"._BOOL.BASEPOS_Req;
      O     "DB_Steps"._BOOL.EMPTY_Req;
      O     "DB_Steps"._BOOL.GET_Req;
      O     "DB_Steps"._BOOL.PUT_Req;
      );
      L     S5T#300MS;
      SD    T 70;
      NOP   0;
      NOP   0;
      NOP   0;
      A     T 70;
      =     "DB_Steps"._BOOL.STEPS_start;
NETWORK
TITLE =
      O     "DB_Steps"._BOOL.STEPS_start;
      O     "DB_ComGateway".FM.CleareOrder;
      ON    "ModeAuto";
      R     "DB_Steps"._BOOL.GET_Finished;
NETWORK
TITLE = reset step sequences
      ON    "ModeAuto";
      O     "DB_ComGateway".FM.CleareOrder;
      =     L 35.0;
      A     L 35.0;
      JNB   _019;
      L     0;
      T     "DB_Steps"._INT.BASEPOS_Steps;
_019: NOP   0;
      A     L 35.0;
      JNB   _01a;
      L     0;
      T     "DB_Steps"._INT.EMPTY_Steps;
_01a: NOP   0;
      A     L 35.0;
      JNB   _01b;
      L     0;
      T     "DB_Steps"._INT.GET_Steps;
_01b: NOP   0;
      A     L 35.0;
      JNB   _01c;
      L     0;
      T     "DB_Steps"._INT.PUT_Steps;
_01c: NOP   0;
